KUKA KRL program: MyProgram_280().src

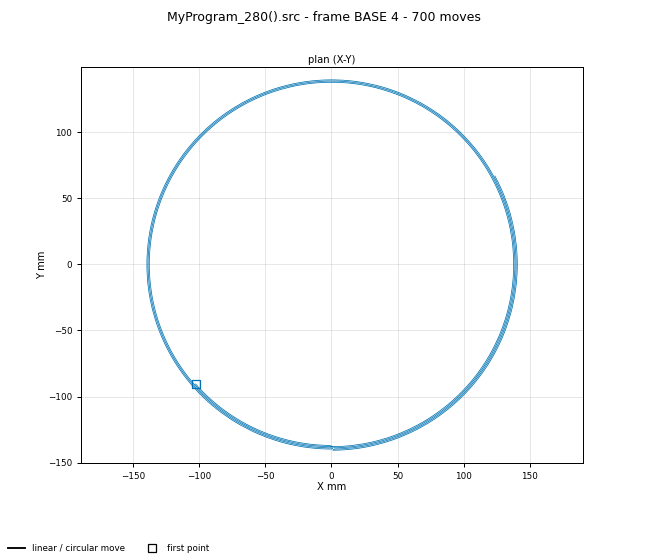
[picture p0: tool path of MyProgram_280().src in frame BASE 4, 700 of 700 moves have a stored position in this frame; points joined in program order, loops and branches not executed]
&ACCESS RVP
&REL 1
&PARAM TEMPLATE = C:\KRC\Roboter\Template\vorgabe
&PARAM EDITMASK = *
DEF MyProgram_280()
; ---- Setting reference (Base) ----
$BASE = BASE_DATA[4]

; --------------------------
; ---- Setting tool (TCP) ----
$TOOL = TOOL_DATA[3]
; --------------------------

$VEL.CP = VEL_APROX_PRINT
Startdeposition()
$VEL.CP = VEL_PRINT
LIN {X -102.883,Y -90.5499,Z 173,A -135.8281,B 8.3337,C 0.3369,E1 8.2218,E2 227.3937} C_DIS
LIN {X -99.9012,Y -93.8294,Z 173,A -133.9555,B 8.3335,C 0.3404,E1 8.2253,E2 225.5192} C_DIS
LIN {X -96.8965,Y -96.9297,Z 173,A -132.2443,B 8.3333,C 0.3455,E1 8.2287,E2 223.8206} C_DIS
LIN {X -93.9619,Y -99.7762,Z 173,A -130.464,B 8.3333,C 0.3476,E1 8.2323,E2 222.0316} C_DIS
LIN {X -90.696,Y -102.7539,Z 173,A -128.5932,B 8.3331,C 0.3506,E1 8.2362,E2 220.1583} C_DIS
LIN {X -87.7529,Y -105.2794,Z 173,A -126.8961,B 8.3331,C 0.3523,E1 8.2398,E2 218.452} C_DIS
LIN {X -84.2582,Y -108.0963,Z 173,A -125.0334,B 8.3329,C 0.3557,E1 8.2439,E2 216.5914} C_DIS
LIN {X -80.7877,Y -110.7143,Z 173,A -123.206,B 8.3328,C 0.3585,E1 8.248,E2 214.763} C_DIS
LIN {X -77.8003,Y -112.8331,Z 173,A -121.6319,B 8.3328,C 0.3602,E1 8.2516,E2 213.1836} C_DIS
LIN {X -74.2625,Y -115.1929,Z 173,A -119.9315,B 8.3325,C 0.3641,E1 8.2556,E2 211.4933} C_DIS
LIN {X -71.2942,Y -117.0532,Z 173,A -118.3313,B 8.3325,C 0.3639,E1 8.2594,E2 209.8758} C_DIS
LIN {X -67.4734,Y -119.2963,Z 173,A -116.5707,B 8.3324,C 0.368,E1 8.2636,E2 208.1271} C_DIS
LIN {X -64.4842,Y -120.9384,Z 173,A -115.1531,B 8.3323,C 0.3699,E1 8.2671,E2 206.7105} C_DIS
LIN {X -60.9886,Y -122.7359,Z 173,A -113.5525,B 8.3322,C 0.3726,E1 8.2711,E2 205.1153} C_DIS
LIN {X -57.8973,Y -124.2242,Z 173,A -112.0982,B 8.3322,C 0.3739,E1 8.2748,E2 203.6584} C_DIS
LIN {X -55.176,Y -125.4588,Z 173,A -110.7127,B 8.3322,C 0.3729,E1 8.2783,E2 202.2555} C_DIS
LIN {X -51.7787,Y -126.8971,Z 173,A -109.3505,B 8.332,C 0.3776,E1 8.2818,E2 200.9162} C_DIS
LIN {X -48.8661,Y -128.0485,Z 173,A -107.9192,B 8.332,C 0.3767,E1 8.2856,E2 199.4691} C_DIS
LIN {X -45.4055,Y -129.3145,Z 173,A -106.4697,B 8.3319,C 0.3796,E1 8.2893,E2 198.031} C_DIS
LIN {X -42.2502,Y -130.3796,Z 173,A -104.991,B 8.3319,C 0.3792,E1 8.2933,E2 196.541} C_DIS
LIN {X -39.0567,Y -131.3717,Z 173,A -103.5138,B 8.3319,C 0.3788,E1 8.2973,E2 195.0534} C_DIS
LIN {X -35.5511,Y -132.3624,Z 173,A -102.2773,B 8.3316,C 0.3849,E1 8.3005,E2 193.8532} C_DIS
LIN {X -32.916,Y -133.0445,Z 173,A -100.8373,B 8.3318,C 0.3802,E1 8.3045,E2 192.3743} C_DIS
LIN {X -29.7209,Y -133.7945,Z 173,A -99.4335,B 8.3318,C 0.3802,E1 8.3083,E2 190.966} C_DIS
LIN {X -25.9901,Y -134.5668,Z 173,A -98.0033,B 8.3317,C 0.3839,E1 8.3122,E2 189.5562} C_DIS
LIN {X -23.3494,Y -135.0523,Z 173,A -96.7469,B 8.3317,C 0.382,E1 8.3157,E2 188.2824} C_DIS
LIN {X -19.5757,Y -135.6484,Z 173,A -95.4567,B 8.3315,C 0.388,E1 8.3192,E2 187.0309} C_DIS
LIN {X -16.7714,Y -136.0246,Z 173,A -94.0487,B 8.3316,C 0.3842,E1 8.3231,E2 185.5937} C_DIS
LIN {X -13.2633,Y -136.4104,Z 173,A -92.8033,B 8.3314,C 0.3887,E1 8.3265,E2 184.3772} C_DIS
LIN {X -10.7558,Y -136.6332,Z 173,A -91.5229,B 8.3316,C 0.3847,E1 8.3302,E2 183.0672} C_DIS
LIN {X -7.653,Y -136.842,Z 173,A -90.2245,B 8.3316,C 0.3847,E1 8.3338,E2 181.7685} C_DIS
LIN {X -4.3301,Y -136.9863,Z 173,A -88.9268,B 8.3316,C 0.3865,E1 8.3374,E2 180.482} C_DIS
LIN {X -1.277,Y -137.0488,Z 173,A -87.465,B 8.3317,C 0.3829,E1 8.3415,E2 178.9959} C_DIS
LIN {X -1.277,Y -137.0488,Z 173,A -87.465,B 8.3317,C 0.3829,E1 8.3415,E2 178.9959} C_DIS
Enddeposition()
LIN {X 0.9792,Y -137.9557,Z 173,A -86.7312,B 8.287,C 0.3922,E1 8.2992,E2 178.3349} C_DIS
Startdeposition()
$VEL.CP = VEL_PRINT
LIN {X -2.0656,Y -137.947,Z 173,A -88.4524,B 8.2866,C 0.4008,E1 8.2942,E2 180.1156} C_DIS
LIN {X -5.8121,Y -137.8404,Z 173,A -89.9694,B 8.2866,C 0.4001,E1 8.29,E2 181.6282} C_DIS
LIN {X -9.6417,Y -137.6255,Z 173,A -91.5436,B 8.2866,C 0.3997,E1 8.2856,E2 183.2007} C_DIS
LIN {X -13.0454,Y -137.3441,Z 173,A -93.0201,B 8.2866,C 0.4006,E1 8.2815,E2 184.6851} C_DIS
LIN {X -16.3304,Y -136.9922,Z 173,A -94.7606,B 8.2863,C 0.407,E1 8.2765,E2 186.4732} C_DIS
LIN {X -20.1888,Y -136.4786,Z 173,A -95.9522,B 8.2867,C 0.3988,E1 8.2734,E2 187.6112} C_DIS
LIN {X -25.0424,Y -135.6715,Z 173,A -98.129,B 8.2867,C 0.4005,E1 8.2673,E2 189.8057} C_DIS
LIN {X -29.337,Y -134.8069,Z 173,A -99.8936,B 8.2867,C 0.3986,E1 8.2625,E2 191.5637} C_DIS
LIN {X -35.9245,Y -133.2031,Z 173,A -102.8001,B 8.2867,C 0.3986,E1 8.2546,E2 194.4825} C_DIS
LIN {X -39.9371,Y -132.0557,Z 173,A -104.3094,B 8.287,C 0.3934,E1 8.2506,E2 195.9636} C_DIS
LIN {X -43.1517,Y -131.0405,Z 173,A -105.8881,B 8.2869,C 0.3955,E1 8.2464,E2 197.5653} C_DIS
LIN {X -46.4079,Y -129.9228,Z 173,A -107.325,B 8.2869,C 0.3944,E1 8.2426,E2 199.0034} C_DIS
LIN {X -49.8097,Y -128.6564,Z 173,A -108.7224,B 8.2871,C 0.3911,E1 8.239,E2 200.3869} C_DIS
LIN {X -52.8849,Y -127.4234,Z 173,A -110.0787,B 8.2871,C 0.3894,E1 8.2355,E2 201.7409} C_DIS
LIN {X -55.7193,Y -126.2111,Z 173,A -111.6175,B 8.2871,C 0.3926,E1 8.2314,E2 203.3128} C_DIS
LIN {X -59.2158,Y -124.6074,Z 173,A -113.0992,B 8.2871,C 0.3888,E1 8.2277,E2 204.7798} C_DIS
LIN {X -62.027,Y -123.2334,Z 173,A -114.479,B 8.2871,C 0.3886,E1 8.2242,E2 206.1699} C_DIS
LIN {X -67.6249,Y -120.2533,Z 173,A -117.118,B 8.2873,C 0.3854,E1 8.2178,E2 208.8095} C_DIS
LIN {X -71.5832,Y -117.9401,Z 173,A -119.0316,B 8.2875,C 0.3829,E1 8.2132,E2 210.7242} C_DIS
LIN {X -75.3846,Y -115.5476,Z 173,A -120.9173,B 8.2875,C 0.3805,E1 8.2087,E2 212.6123} C_DIS
LIN {X -79.0785,Y -113.0517,Z 173,A -122.5617,B 8.2879,C 0.3742,E1 8.205,E2 214.2301} C_DIS
LIN {X -82.8628,Y -110.3079,Z 173,A -124.8045,B 8.2878,C 0.3761,E1 8.1999,E2 216.511} C_DIS
LIN {X -86.4464,Y -107.5223,Z 173,A -126.6718,B 8.2879,C 0.3725,E1 8.1958,E2 218.3757} C_DIS
LIN {X -89.7939,Y -104.7432,Z 173,A -128.5379,B 8.288,C 0.3703,E1 8.1918,E2 220.2489} C_DIS
LIN {X -93.0689,Y -101.8446,Z 173,A -130.3846,B 8.2882,C 0.3674,E1 8.1879,E2 222.099} C_DIS
LIN {X -96.4499,Y -98.648,Z 173,A -132.3135,B 8.2883,C 0.3636,E1 8.1841,E2 224.0269} C_DIS
LIN {X -99.3487,Y -95.7284,Z 173,A -133.9538,B 8.2885,C 0.3591,E1 8.1809,E2 225.658} C_DIS
LIN {X -102.0619,Y -92.8298,Z 173,A -135.8247,B 8.2885,C 0.3593,E1 8.1773,E2 227.5564} C_DIS
LIN {X -105.4509,Y -88.9619,Z 173,A -137.8991,B 8.2887,C 0.3538,E1 8.1735,E2 229.6222} C_DIS
LIN {X -108.3711,Y -85.3799,Z 173,A -139.8171,B 8.2889,C 0.3496,E1 8.1702,E2 231.5393} C_DIS
LIN {X -111.0969,Y -81.8015,Z 173,A -141.7145,B 8.2891,C 0.3458,E1 8.167,E2 233.4395} C_DIS
LIN {X -113.8226,Y -77.9641,Z 173,A -143.6412,B 8.2893,C 0.3408,E1 8.1639,E2 235.3618} C_DIS
LIN {X -116.0236,Y -74.6499,Z 173,A -145.3906,B 8.2893,C 0.3385,E1 8.1612,E2 237.1226} C_DIS
LIN {X -118.3482,Y -70.9068,Z 173,A -147.2546,B 8.2895,C 0.3346,E1 8.1585,E2 238.9899} C_DIS
LIN {X -120.7103,Y -66.8058,Z 173,A -148.9434,B 8.2899,C 0.3254,E1 8.1562,E2 240.6428} C_DIS
LIN {X -122.6542,Y -63.1648,Z 173,A -150.9243,B 8.2899,C 0.3252,E1 8.1536,E2 242.6563} C_DIS
LIN {X -124.3506,Y -59.7532,Z 173,A -152.4716,B 8.2901,C 0.3206,E1 8.1517,E2 244.1982} C_DIS
LIN {X -125.9172,Y -56.3763,Z 173,A -154.0438,B 8.2902,C 0.317,E1 8.1499,E2 245.7727} C_DIS
LIN {X -127.6592,Y -52.3184,Z 173,A -156.1711,B 8.2902,C 0.3167,E1 8.1476,E2 247.9356} C_DIS
LIN {X -129.6287,Y -47.2236,Z 173,A -158.1322,B 8.2906,C 0.306,E1 8.1457,E2 249.8567} C_DIS
LIN {X -131.0791,Y -43.0356,Z 173,A -160.2173,B 8.2906,C 0.3047,E1 8.1438,E2 251.9711} C_DIS
LIN {X -132.2357,Y -39.339,Z 173,A -161.6204,B 8.291,C 0.2972,E1 8.1426,E2 253.3474} C_DIS
LIN {X -133.2526,Y -35.7387,Z 173,A -163.1895,B 8.291,C 0.2931,E1 8.1415,E2 254.9171} C_DIS
LIN {X -134.083,Y -32.4849,Z 173,A -164.7412,B 8.2911,C 0.2916,E1 8.1404,E2 256.4875} C_DIS
LIN {X -134.8591,Y -29.0949,Z 173,A -166.1771,B 8.2913,C 0.2874,E1 8.1395,E2 257.9212} C_DIS
LIN {X -135.4963,Y -25.9666,Z 173,A -167.5733,B 8.2913,C 0.2847,E1 8.1388,E2 259.3251} C_DIS
LIN {X -136.1899,Y -22.0519,Z 173,A -169.348,B 8.2915,C 0.2819,E1 8.1379,E2 261.1141} C_DIS
LIN {X -136.7862,Y -17.9745,Z 173,A -170.9916,B 8.2917,C 0.276,E1 8.1373,E2 262.7477} C_DIS
LIN {X -137.1338,Y -15.0987,Z 173,A -172.2937,B 8.2917,C 0.274,E1 8.1369,E2 264.0611} C_DIS
LIN {X -137.5557,Y -10.5972,Z 173,A -174.1761,B 8.2919,C 0.2687,E1 8.1364,E2 265.9426} C_DIS
LIN {X -137.7677,Y -7.334,Z 173,A -175.3466,B 8.2921,C 0.262,E1 8.1362,E2 267.0885} C_DIS
LIN {X -137.9073,Y -3.8946,Z 173,A -176.7229,B 8.2923,C 0.2571,E1 8.1362,E2 268.4568} C_DIS
LIN {X -137.9604,Y -0.8702,Z 173,A -178.3723,B 8.2923,C 0.2593,E1 8.136,E2 270.1542} C_DIS
LIN {X -137.9142,Y 3.6454,Z 173,A 179.8464,B 8.2924,C 0.2525,E1 8.1361,E2 271.922} C_DIS
LIN {X -137.7534,Y 7.6193,Z 173,A 178.0993,B 8.2925,C 0.2491,E1 8.1364,E2 273.6796} C_DIS
LIN {X -137.5136,Y 11.1273,Z 173,A 176.677,B 8.2927,C 0.2444,E1 8.1367,E2 275.0958} C_DIS
LIN {X -137.266,Y 13.8585,Z 173,A 175.3981,B 8.2927,C 0.2432,E1 8.137,E2 276.391} C_DIS
LIN {X -136.7966,Y 17.8947,Z 173,A 173.84,B 8.2929,C 0.2364,E1 8.1375,E2 277.9314} C_DIS
LIN {X -136.2081,Y 21.9404,Z 173,A 171.938,B 8.2929,C 0.2345,E1 8.1384,E2 279.8571} C_DIS
LIN {X -135.5693,Y 25.5851,Z 173,A 170.1954,B 8.2929,C 0.2332,E1 8.1393,E2 281.6236} C_DIS
LIN {X -134.8756,Y 29.0186,Z 173,A 169.0835,B 8.2932,C 0.224,E1 8.1399,E2 282.6917} C_DIS
LIN {X -134.1832,Y 32.0691,Z 173,A 167.8519,B 8.2934,C 0.2193,E1 8.1406,E2 283.9137} C_DIS
LIN {X -133.5479,Y 34.626,Z 173,A 166.4523,B 8.2934,C 0.2208,E1 8.1416,E2 285.3501} C_DIS
LIN {X -132.4614,Y 38.568,Z 173,A 164.9416,B 8.2935,C 0.2133,E1 8.1428,E2 286.8359} C_DIS
LIN {X -131.4885,Y 41.7647,Z 173,A 163.4664,B 8.2935,C 0.2107,E1 8.144,E2 288.3205} C_DIS
LIN {X -130.3861,Y 45.0881,Z 173,A 162.0908,B 8.2937,C 0.2055,E1 8.1452,E2 289.685} C_DIS
LIN {X -129.4148,Y 47.8086,Z 173,A 160.87,B 8.2937,C 0.2026,E1 8.1464,E2 290.9072} C_DIS
LIN {X -128.0471,Y 51.356,Z 173,A 159.1779,B 8.2938,C 0.2,E1 8.1481,E2 292.6117} C_DIS
LIN {X -126.8766,Y 54.1862,Z 173,A 157.9737,B 8.2939,C 0.1956,E1 8.1494,E2 293.8063} C_DIS
LIN {X -125.338,Y 57.6533,Z 173,A 156.3034,B 8.294,C 0.1928,E1 8.1513,E2 295.4868} C_DIS
LIN {X -124.0777,Y 60.3222,Z 173,A 154.9133,B 8.294,C 0.1921,E1 8.153,E2 296.8959} C_DIS
LIN {X -122.3229,Y 63.8018,Z 173,A 153.4395,B 8.2942,C 0.1857,E1 8.1549,E2 298.3502} C_DIS
LIN {X -119.4454,Y 69.042,Z 173,A 150.8189,B 8.2942,C 0.1815,E1 8.1585,E2 300.9854} C_DIS
LIN {X -117.4741,Y 72.3455,Z 173,A 149.3691,B 8.2944,C 0.1753,E1 8.1605,E2 302.4155} C_DIS
LIN {X -115.4763,Y 75.4944,Z 173,A 147.5373,B 8.2944,C 0.1758,E1 8.1634,E2 304.2805} C_DIS
LIN {X -112.8589,Y 79.353,Z 173,A 145.5986,B 8.2944,C 0.1711,E1 8.1664,E2 306.2175} C_DIS
LIN {X -108.0056,Y 85.8415,Z 173,A 142.2322,B 8.2946,C 0.1634,E1 8.1721,E2 309.5808} C_DIS
LIN {X -105.3842,Y 89.0411,Z 173,A 140.4942,B 8.2947,C 0.1598,E1 8.1752,E2 311.3197} C_DIS
LIN {X -102.6871,Y 92.1376,Z 173,A 138.6772,B 8.2947,C 0.1578,E1 8.1786,E2 313.1487} C_DIS
LIN {X -99.6124,Y 95.4535,Z 173,A 136.8822,B 8.2948,C 0.1525,E1 8.182,E2 314.9317} C_DIS
LIN {X -96.9458,Y 98.1614,Z 173,A 135.2534,B 8.2948,C 0.1501,E1 8.1852,E2 316.5652} C_DIS
LIN {X -94.5977,Y 100.4254,Z 173,A 133.9095,B 8.2949,C 0.1472,E1 8.1879,E2 317.9065} C_DIS
LIN {X -91.4098,Y 103.3355,Z 173,A 132.0978,B 8.2949,C 0.144,E1 8.1917,E2 319.7189} C_DIS
LIN {X -88.4225,Y 105.9035,Z 173,A 130.3946,B 8.295,C 0.142,E1 8.1953,E2 321.4288} C_DIS
LIN {X -84.6977,Y 108.9051,Z 173,A 128.1797,B 8.295,C 0.142,E1 8.2003,E2 323.6698} C_DIS
LIN {X -82.0737,Y 110.8966,Z 173,A 126.9549,B 8.2951,C 0.1373,E1 8.203,E2 324.8759} C_DIS
LIN {X -78.2616,Y 113.6185,Z 173,A 125.0033,B 8.2951,C 0.1341,E1 8.2074,E2 326.8265} C_DIS
LIN {X -74.5584,Y 116.0821,Z 173,A 123.1927,B 8.2952,C 0.1306,E1 8.2116,E2 328.631} C_DIS
LIN {X -70.8901,Y 118.3582,Z 173,A 121.4157,B 8.2952,C 0.1276,E1 8.2159,E2 330.4046} C_DIS
LIN {X -66.2435,Y 121.0199,Z 173,A 119.0875,B 8.2952,C 0.1261,E1 8.2216,E2 332.7437} C_DIS
LIN {X -62.8343,Y 122.8224,Z 173,A 117.4404,B 8.2953,C 0.1247,E1 8.2256,E2 334.3949} C_DIS
LIN {X -58.5256,Y 124.9346,Z 173,A 115.4281,B 8.2953,C 0.1225,E1 8.2307,E2 336.4081} C_DIS
LIN {X -54.0934,Y 126.9167,Z 173,A 113.4525,B 8.2953,C 0.1195,E1 8.2358,E2 338.3772} C_DIS
LIN {X -50.0528,Y 128.5619,Z 173,A 111.7351,B 8.2954,C 0.1159,E1 8.2402,E2 340.0816} C_DIS
LIN {X -44.4017,Y 130.6241,Z 173,A 109.0787,B 8.2954,C 0.1161,E1 8.2472,E2 342.7556} C_DIS
LIN {X -40.5455,Y 131.8695,Z 173,A 107.5266,B 8.2954,C 0.1124,E1 8.2513,E2 344.2905} C_DIS
LIN {X -37.5348,Y 132.7583,Z 173,A 106.3779,B 8.2955,C 0.1087,E1 8.2543,E2 345.4192} C_DIS
LIN {X -34.2608,Y 133.6405,Z 173,A 104.8017,B 8.2955,C 0.1105,E1 8.2586,E2 347.0152} C_DIS
LIN {X -31.2296,Y 134.3819,Z 173,A 103.3807,B 8.2955,C 0.1118,E1 8.2625,E2 348.4506} C_DIS
LIN {X -27.6928,Y 135.1542,Z 173,A 102.1194,B 8.2955,C 0.1067,E1 8.2659,E2 349.6813} C_DIS
LIN {X -24.149,Y 135.8321,Z 173,A 100.5924,B 8.2955,C 0.1064,E1 8.2701,E2 351.2109} C_DIS
LIN {X -18.9902,Y 136.6499,Z 173,A 98.2921,B 8.2955,C 0.1077,E1 8.2765,E2 353.5262} C_DIS
LIN {X -15.1944,Y 137.1235,Z 173,A 96.2626,B 8.2955,C 0.1148,E1 8.2823,E2 355.6085} C_DIS
LIN {X -11.0614,Y 137.5191,Z 173,A 94.0381,B 8.2953,C 0.123,E1 8.2886,E2 357.8926} C_DIS
LIN {X -4.2782,Y 137.8966,Z 173,A 92.1554,B 8.2956,C 0.1063,E1 8.2936,E2 359.66} C_DIS
LIN {X 2.4377,Y 137.9408,Z 173,A 89.4986,B 8.2956,C 0.1039,E1 8.3009,E2 362.2993} C_DIS
LIN {X 9.6118,Y 137.6276,Z 173,A 86.5437,B 8.2956,C 0.1039,E1 8.3092,E2 365.2498} C_DIS
LIN {X 14.0894,Y 137.2425,Z 173,A 84.2938,B 8.2955,C 0.1112,E1 8.3156,E2 367.5462} C_DIS
LIN {X 17.8918,Y 136.797,Z 173,A 82.5683,B 8.2955,C 0.1142,E1 8.3204,E2 369.2876} C_DIS
LIN {X 21.6437,Y 136.2548,Z 173,A 81.2679,B 8.2955,C 0.1099,E1 8.3239,E2 370.5541} C_DIS
LIN {X 25.8341,Y 135.5216,Z 173,A 79.8227,B 8.2955,C 0.1049,E1 8.3277,E2 371.9592} C_DIS
LIN {X 28.7334,Y 134.9372,Z 173,A 77.9527,B 8.2955,C 0.1174,E1 8.3331,E2 373.9076} C_DIS
LIN {X 32.6672,Y 134.0391,Z 173,A 76.6406,B 8.2955,C 0.1118,E1 8.3365,E2 375.1749} C_DIS
LIN {X 36.9153,Y 132.9316,Z 173,A 75.1032,B 8.2955,C 0.1078,E1 8.3406,E2 376.6766} C_DIS
LIN {X 40.2181,Y 131.9697,Z 173,A 73.4973,B 8.2955,C 0.1123,E1 8.3449,E2 378.3042} C_DIS
LIN {X 43.4246,Y 130.9496,Z 173,A 72.0922,B 8.2955,C 0.1137,E1 8.3486,E2 379.71} C_DIS
LIN {X 46.7016,Y 129.8169,Z 173,A 70.6385,B 8.2955,C 0.1153,E1 8.3525,E2 381.1652} C_DIS
LIN {X 49.8442,Y 128.643,Z 173,A 69.3066,B 8.2955,C 0.1155,E1 8.3559,E2 382.4895} C_DIS
LIN {X 52.8129,Y 127.4535,Z 173,A 67.8602,B 8.2954,C 0.1192,E1 8.3597,E2 383.9503} C_DIS
LIN {X 56.2817,Y 125.9596,Z 173,A 66.4297,B 8.2954,C 0.1184,E1 8.3633,E2 385.3637} C_DIS
LIN {X 58.8172,Y 124.7978,Z 173,A 65.1493,B 8.2954,C 0.1221,E1 8.3666,E2 386.6592} C_DIS
LIN {X 64.1268,Y 122.1522,Z 173,A 62.8294,B 8.2954,C 0.1225,E1 8.3724,E2 388.9613} C_DIS
LIN {X 67.8596,Y 120.1214,Z 173,A 60.9316,B 8.2953,C 0.1276,E1 8.377,E2 390.8756} C_DIS
LIN {X 71.4457,Y 118.0233,Z 173,A 59.168,B 8.2953,C 0.1308,E1 8.3813,E2 392.644} C_DIS
LIN {X 75.4355,Y 115.5145,Z 173,A 56.7358,B 8.295,C 0.1431,E1 8.3871,E2 395.1347} C_DIS
LIN {X 79.858,Y 112.5026,Z 173,A 55.1002,B 8.2951,C 0.1353,E1 8.3907,E2 396.6986} C_DIS
LIN {X 83.4863,Y 109.837,Z 173,A 53.2184,B 8.2951,C 0.1387,E1 8.3949,E2 398.5822} C_DIS
LIN {X 87.0974,Y 106.9957,Z 173,A 51.3463,B 8.2951,C 0.1414,E1 8.399,E2 400.4502} C_DIS
LIN {X 90.4066,Y 104.2151,Z 173,A 49.7304,B 8.2951,C 0.1412,E1 8.4023,E2 402.0444} C_DIS
LIN {X 92.9479,Y 101.9548,Z 173,A 48.199,B 8.295,C 0.1463,E1 8.4056,E2 403.5909} C_DIS
LIN {X 95.0442,Y 100.0037,Z 173,A 46.8658,B 8.2949,C 0.1515,E1 8.4083,E2 404.9422} C_DIS
LIN {X 98.5503,Y 96.5496,Z 173,A 44.3971,B 8.2946,C 0.1642,E1 8.4133,E2 407.4639} C_DIS
LIN {X 102.3654,Y 92.4953,Z 173,A 42.7347,B 8.2948,C 0.156,E1 8.4162,E2 409.0471} C_DIS
LIN {X 105.1615,Y 89.303,Z 173,A 41.0308,B 8.2948,C 0.1586,E1 8.4193,E2 410.7443} C_DIS
LIN {X 107.7501,Y 86.1625,Z 173,A 39.4496,B 8.2948,C 0.1602,E1 8.4221,E2 412.3126} C_DIS
LIN {X 110.3043,Y 82.8676,Z 173,A 37.602,B 8.2946,C 0.1665,E1 8.4252,E2 414.1755} C_DIS
LIN {X 112.8049,Y 79.4295,Z 173,A 35.8745,B 8.2946,C 0.1698,E1 8.428,E2 415.8991} C_DIS
LIN {X 115.6759,Y 75.1869,Z 173,A 33.7901,B 8.2944,C 0.174,E1 8.4313,E2 417.9791} C_DIS
LIN {X 117.6682,Y 72.0291,Z 173,A 31.4583,B 8.294,C 0.1939,E1 8.4348,E2 420.4085} C_DIS
LIN {X 120.956,Y 66.3608,Z 173,A 29.5461,B 8.2942,C 0.184,E1 8.4373,E2 422.2221} C_DIS
LIN {X 122.8108,Y 62.8571,Z 173,A 28.056,B 8.2942,C 0.1849,E1 8.4392,E2 423.6936} C_DIS
LIN {X 124.0311,Y 60.4167,Z 173,A 26.7856,B 8.2941,C 0.1907,E1 8.4408,E2 424.9818} C_DIS
LIN {X 125.8177,Y 56.5988,Z 173,A 25.148,B 8.2941,C 0.1929,E1 8.4426,E2 426.6064} C_DIS
LIN {X 127.1655,Y 53.5024,Z 173,A 23.5644,B 8.2938,C 0.2004,E1 8.4444,E2 428.2135} C_DIS
LIN {X 129.0833,Y 48.6934,Z 173,A 21.8115,B 8.2938,C 0.1979,E1 8.4461,E2 429.9182} C_DIS
LIN {X 130.2557,Y 45.4643,Z 173,A 20.3126,B 8.2938,C 0.2033,E1 8.4476,E2 431.4271} C_DIS
LIN {X 131.3571,Y 42.176,Z 173,A 18.8517,B 8.2937,C 0.2076,E1 8.4488,E2 432.8916} C_DIS
LIN {X 132.4689,Y 38.5423,Z 173,A 17.3109,B 8.2936,C 0.2112,E1 8.4501,E2 434.4289} C_DIS
LIN {X 133.5496,Y 34.6192,Z 173,A 15.7227,B 8.2936,C 0.2137,E1 8.4512,E2 436.0056} C_DIS
LIN {X 134.2706,Y 31.7066,Z 173,A 14.363,B 8.2934,C 0.2196,E1 8.4521,E2 437.3805} C_DIS
LIN {X 135.3757,Y 26.5975,Z 173,A 12.2298,B 8.2932,C 0.225,E1 8.4533,E2 439.5108} C_DIS
LIN {X 136.0321,Y 22.9972,Z 173,A 10.7781,B 8.2932,C 0.2278,E1 8.454,E2 440.9551} C_DIS
LIN {X 136.4964,Y 20.0641,Z 173,A 9.58,B 8.2931,C 0.2306,E1 8.4545,E2 442.1497} C_DIS
LIN {X 136.9545,Y 16.6463,Z 173,A 8.332,B 8.2931,C 0.2308,E1 8.455,E2 443.3757} C_DIS
LIN {X 137.4651,Y 11.7013,Z 173,A 6.3071,B 8.2929,C 0.2359,E1 8.4555,E2 445.3974} C_DIS
LIN {X 137.8923,Y 4.4322,Z 173,A 2.4349,B 8.2921,C 0.2626,E1 8.456,E2 449.3788} C_DIS
LIN {X 137.9561,Y -1.5094,Z 173,A 0.8012,B 8.2924,C 0.2521,E1 8.456,E2 450.9101} C_DIS
LIN {X 137.657,Y -9.1992,Z 173,A -2.2907,B 8.2922,C 0.2591,E1 8.4557,E2 453.9919} C_DIS
LIN {X 136.9661,Y -16.5491,Z 173,A -4.9984,B 8.2922,C 0.2603,E1 8.455,E2 456.657} C_DIS
LIN {X 136.1629,Y -22.2132,Z 173,A -7.9334,B 8.2916,C 0.2791,E1 8.4537,E2 459.6656} C_DIS
LIN {X 135.038,Y -28.2635,Z 173,A -10.2159,B 8.2916,C 0.2806,E1 8.4525,E2 461.9159} C_DIS
LIN {X 134.3943,Y -31.1752,Z 173,A -11.5694,B 8.2913,C 0.2866,E1 8.4517,E2 463.2852} C_DIS
LIN {X 133.5485,Y -34.6235,Z 173,A -12.9835,B 8.2913,C 0.2895,E1 8.4507,E2 464.6932} C_DIS
LIN {X 132.6447,Y -37.9395,Z 173,A -14.4161,B 8.2911,C 0.2936,E1 8.4496,E2 466.1278} C_DIS
LIN {X 131.5129,Y -41.6883,Z 173,A -15.9147,B 8.2911,C 0.2954,E1 8.4484,E2 467.6118} C_DIS
LIN {X 130.3865,Y -45.087,Z 173,A -17.3284,B 8.2909,C 0.2979,E1 8.4471,E2 469.0177} C_DIS
LIN {X 129.4055,Y -47.8333,Z 173,A -18.4578,B 8.2909,C 0.2995,E1 8.4461,E2 470.1379} C_DIS
LIN {X 127.8905,Y -51.7446,Z 173,A -20.2536,B 8.2907,C 0.3054,E1 8.4442,E2 471.9424} C_DIS
LIN {X 126.6647,Y -54.6763,Z 173,A -21.5571,B 8.2905,C 0.3086,E1 8.4428,E2 473.2451} C_DIS
LIN {X 123.554,Y -61.3839,Z 173,A -24.5387,B 8.2903,C 0.3149,E1 8.4393,E2 476.2185} C_DIS
LIN {X 121.8158,Y -64.7676,Z 173,A -26.1934,B 8.2901,C 0.3206,E1 8.4371,E2 477.8844} C_DIS
LIN {X 119.8061,Y -68.414,Z 173,A -27.9228,B 8.2899,C 0.3251,E1 8.4348,E2 479.6156} C_DIS
LIN {X 117.8429,Y -71.7423,Z 173,A -29.9468,B 8.2894,C 0.3379,E1 8.4318,E2 481.6946} C_DIS
LIN {X 115.366,Y -75.6618,Z 173,A -31.3709,B 8.2896,C 0.3322,E1 8.4297,E2 483.0569} C_DIS
LIN {X 113.106,Y -79.0005,Z 173,A -32.9855,B 8.2896,C 0.335,E1 8.4271,E2 484.6655} C_DIS
LIN {X 110.7876,Y -82.22,Z 173,A -34.5935,B 8.2894,C 0.3382,E1 8.4245,E2 486.2702} C_DIS
LIN {X 107.439,Y -86.5497,Z 173,A -36.9137,B 8.2891,C 0.3445,E1 8.4205,E2 488.5987} C_DIS
LIN {X 104.8112,Y -89.7149,Z 173,A -38.6292,B 8.289,C 0.3485,E1 8.4174,E2 490.3168} C_DIS
LIN {X 102.4431,Y -92.4097,Z 173,A -40.926,B 8.2881,C 0.3685,E1 8.4129,E2 492.7174} C_DIS
LIN {X 97.7231,Y -97.387,Z 173,A -42.6543,B 8.2888,C 0.3515,E1 8.4098,E2 494.3062} C_DIS
LIN {X 92.825,Y -102.0663,Z 173,A -45.9549,B 8.2882,C 0.3673,E1 8.403,E2 497.6718} C_DIS
LIN {X 90.0018,Y -104.5639,Z 173,A -47.4217,B 8.2882,C 0.3684,E1 8.3999,E2 499.1276} C_DIS
LIN {X 87.4209,Y -106.7314,Z 173,A -48.5305,B 8.2882,C 0.3652,E1 8.3976,E2 500.2006} C_DIS
LIN {X 80.5503,Y -112.0076,Z 173,A -52.2363,B 8.2879,C 0.374,E1 8.3893,E2 503.9236} C_DIS
LIN {X 76.5129,Y -114.8032,Z 173,A -54.1437,B 8.2879,C 0.3748,E1 8.3849,E2 505.8159} C_DIS
LIN {X 72.2616,Y -117.5256,Z 173,A -56.4554,B 8.2875,C 0.3825,E1 8.3794,E2 508.1569} C_DIS
LIN {X 69.3793,Y -119.2501,Z 173,A -57.651,B 8.2875,C 0.3807,E1 8.3765,E2 509.3283} C_DIS
LIN {X 65.4205,Y -121.4667,Z 173,A -59.5615,B 8.2875,C 0.3841,E1 8.3718,E2 511.2438} C_DIS
LIN {X 61.4938,Y -123.4998,Z 173,A -61.2232,B 8.2875,C 0.3832,E1 8.3678,E2 512.8846} C_DIS
LIN {X 58.8169,Y -124.798,Z 173,A -62.6357,B 8.2872,C 0.3884,E1 8.3641,E2 514.3209} C_DIS
LIN {X 52.5865,Y -127.548,Z 173,A -65.1704,B 8.2873,C 0.3861,E1 8.3577,E2 516.8201} C_DIS
LIN {X 47.5517,Y -129.5104,Z 173,A -67.5563,B 8.2871,C 0.3915,E1 8.3515,E2 519.226} C_DIS
LIN {X 42.1045,Y -131.38,Z 173,A -69.8552,B 8.2871,C 0.3921,E1 8.3454,E2 521.5147} C_DIS
LIN {X 39.0329,Y -132.3253,Z 173,A -71.1777,B 8.287,C 0.3932,E1 8.3419,E2 522.8366} C_DIS
LIN {X 36.1751,Y -133.1363,Z 173,A -72.5335,B 8.2868,C 0.3966,E1 8.3382,E2 524.209} C_DIS
LIN {X 31.3763,Y -134.3483,Z 173,A -74.5549,B 8.2868,C 0.3976,E1 8.3327,E2 526.2273} C_DIS
LIN {X 27.4863,Y -135.1962,Z 173,A -75.9085,B 8.287,C 0.393,E1 8.3291,E2 527.5435} C_DIS
LIN {X 24.6497,Y -135.7425,Z 173,A -77.4053,B 8.2867,C 0.3995,E1 8.3249,E2 529.0792} C_DIS
LIN {X 16.0145,Y -137.0299,Z 173,A -81.034,B 8.2866,C 0.4015,E1 8.3149,E2 532.7105} C_DIS
LIN {X 11.9861,Y -137.441,Z 173,A -82.6646,B 8.2866,C 0.4012,E1 8.3103,E2 534.3354} C_DIS
LIN {X 7.7255,Y -137.7478,Z 173,A -84.4968,B 8.2866,C 0.4028,E1 8.3052,E2 536.1761} C_DIS
LIN {X 4.1448,Y -137.9003,Z 173,A -85.8866,B 8.2866,C 0.4013,E1 8.3013,E2 537.554} C_DIS
LIN {X 0.9792,Y -137.9557,Z 173,A -86.7279,B 8.287,C 0.3927,E1 8.2992,E2 538.3348} C_DIS
Enddeposition()
LIN {X 0.9792,Y -137.9557,Z 173,A -86.7279,B 8.287,C 0.3927,E1 8.2992,E2 538.3348} C_DIS
Startdeposition()
$VEL.CP = VEL_PRINT
LIN {X 2.7915,Y -138.8436,Z 173,A -85.7711,B 8.2411,C 0.3941,E1 8.256,E2 537.3975} C_DIS
LIN {X 6.4638,Y -138.7212,Z 173,A -84.1933,B 8.2411,C 0.3925,E1 8.2604,E2 535.8108} C_DIS
LIN {X 10.1394,Y -138.5001,Z 173,A -82.7319,B 8.2411,C 0.3932,E1 8.2645,E2 534.3561} C_DIS
LIN {X 13.6741,Y -138.1964,Z 173,A -81.1883,B 8.2412,C 0.3911,E1 8.2688,E2 532.8013} C_DIS
LIN {X 18.8142,Y -137.5924,Z 173,A -78.6523,B 8.2416,C 0.3823,E1 8.276,E2 530.2114} C_DIS
LIN {X 22.9677,Y -136.9581,Z 173,A -77.0567,B 8.2416,C 0.3839,E1 8.2803,E2 528.6328} C_DIS
LIN {X 26.6001,Y -136.3002,Z 173,A -75.9155,B 8.2413,C 0.3904,E1 8.2833,E2 527.5409} C_DIS
LIN {X 30.0295,Y -135.5868,Z 173,A -73.8541,B 8.2419,C 0.3772,E1 8.2892,E2 525.3975} C_DIS
LIN {X 34.8677,Y -134.4238,Z 173,A -72.4296,B 8.2414,C 0.3879,E1 8.2928,E2 524.0543} C_DIS
LIN {X 38.0658,Y -133.5532,Z 173,A -70.9272,B 8.2416,C 0.384,E1 8.2969,E2 522.5333} C_DIS
LIN {X 41.9588,Y -132.3803,Z 173,A -69.0938,B 8.2418,C 0.3793,E1 8.3018,E2 520.6782} C_DIS
LIN {X 45.0896,Y -131.3472,Z 173,A -67.8535,B 8.2418,C 0.3803,E1 8.3051,E2 519.4527} C_DIS
LIN {X 49.7627,Y -129.6495,Z 173,A -66.0832,B 8.2416,C 0.3836,E1 8.3096,E2 517.7177} C_DIS
LIN {X 52.678,Y -128.4938,Z 173,A -64.4049,B 8.242,C 0.3743,E1 8.3141,E2 515.988} C_DIS
LIN {X 55.6978,Y -127.2129,Z 173,A -63.2244,B 8.242,C 0.3761,E1 8.317,E2 514.8291} C_DIS
LIN {X 60.1844,Y -125.1515,Z 173,A -61.2903,B 8.242,C 0.3755,E1 8.3219,E2 512.9067} C_DIS
LIN {X 63.4522,Y -123.5274,Z 173,A -59.7786,B 8.242,C 0.3732,E1 8.3257,E2 511.3931} C_DIS
LIN {X 67.5973,Y -121.3105,Z 173,A -57.8518,B 8.2422,C 0.3706,E1 8.3304,E2 509.4664} C_DIS
LIN {X 74.5256,Y -117.1819,Z 173,A -54.5543,B 8.2424,C 0.3659,E1 8.3383,E2 506.1701} C_DIS
LIN {X 78.0932,Y -114.8348,Z 173,A -52.2595,B 8.243,C 0.3519,E1 8.3437,E2 503.8035} C_DIS
LIN {X 82.3148,Y -111.8471,Z 173,A -50.7958,B 8.2426,C 0.362,E1 8.3469,E2 502.426} C_DIS
LIN {X 85.988,Y -109.0487,Z 173,A -49.0413,B 8.2426,C 0.3616,E1 8.3507,E2 500.6895} C_DIS
LIN {X 88.3689,Y -107.1284,Z 173,A -46.9626,B 8.2434,C 0.3421,E1 8.3554,E2 498.5023} C_DIS
LIN {X 92.5328,Y -103.5529,Z 173,A -45.3364,B 8.243,C 0.351,E1 8.3586,E2 496.958} C_DIS
LIN {X 95.8393,Y -100.5005,Z 173,A -43.5723,B 8.2431,C 0.3491,E1 8.3622,E2 495.2043} C_DIS
LIN {X 98.7491,Y -97.6433,Z 173,A -41.2737,B 8.2438,C 0.3325,E1 8.3669,E2 492.8231} C_DIS
LIN {X 102.3649,Y -93.8452,Z 173,A -39.7632,B 8.2434,C 0.3416,E1 8.3696,E2 491.3963} C_DIS
LIN {X 106.6199,Y -88.9821,Z 173,A -37.1608,B 8.2436,C 0.3369,E1 8.3744,E2 488.7997} C_DIS
LIN {X 109.7793,Y -85.0527,Z 173,A -34.9231,B 8.2439,C 0.3288,E1 8.3783,E2 486.5392} C_DIS
LIN {X 112.6169,Y -81.2589,Z 173,A -33.3124,B 8.2439,C 0.3314,E1 8.3809,E2 484.9715} C_DIS
LIN {X 114.5324,Y -78.5355,Z 173,A -31.7365,B 8.2441,C 0.3238,E1 8.3834,E2 483.3678} C_DIS
LIN {X 117.6555,Y -73.7754,Z 173,A -29.3658,B 8.2444,C 0.3175,E1 8.387,E2 480.992} C_DIS
LIN {X 119.6122,Y -70.5583,Z 173,A -27.8851,B 8.2444,C 0.3151,E1 8.3891,E2 479.5192} C_DIS
LIN {X 121.7969,Y -66.7164,Z 173,A -26.0602,B 8.2446,C 0.3104,E1 8.3916,E2 477.6923} C_DIS
LIN {X 124.274,Y -61.9781,Z 173,A -24.0977,B 8.2446,C 0.3098,E1 8.3941,E2 475.7591} C_DIS
LIN {X 128.1029,Y -53.6155,Z 173,A -20.5421,B 8.2448,C 0.3049,E1 8.3982,E2 472.231} C_DIS
LIN {X 130.1071,Y -48.5503,Z 173,A -18.0246,B 8.2453,C 0.2929,E1 8.4007,E2 469.6764} C_DIS
LIN {X 131.3033,Y -45.216,Z 173,A -16.6116,B 8.2453,C 0.2899,E1 8.402,E2 468.2682} C_DIS
LIN {X 132.3085,Y -42.1835,Z 173,A -15.2854,B 8.2455,C 0.2861,E1 8.4032,E2 466.9397} C_DIS
LIN {X 133.9637,Y -36.5975,Z 173,A -12.7731,B 8.2458,C 0.277,E1 8.4051,E2 464.411} C_DIS
LIN {X 134.9341,Y -32.8311,Z 173,A -11.3133,B 8.2458,C 0.2756,E1 8.4061,E2 462.9684} C_DIS
LIN {X 135.8619,Y -28.7555,Z 173,A -9.0496,B 8.2464,C 0.259,E1 8.4075,E2 460.6328} C_DIS
LIN {X 136.8671,Y -23.5132,Z 173,A -7.5976,B 8.2461,C 0.269,E1 8.4081,E2 459.2763} C_DIS
LIN {X 137.4451,Y -19.8477,Z 173,A -6.2593,B 8.2461,C 0.2688,E1 8.4087,E2 457.9614} C_DIS
LIN {X 138.0126,Y -15.4246,Z 173,A -3.5904,B 8.2468,C 0.2455,E1 8.4096,E2 455.1832} C_DIS
LIN {X 138.4893,Y -10.2868,Z 173,A -2.1849,B 8.2465,C 0.2551,E1 8.4099,E2 453.8697} C_DIS
LIN {X 138.8103,Y -4.1053,Z 173,A 0.1651,B 8.2466,C 0.2521,E1 8.4102,E2 451.5437} C_DIS
LIN {X 138.8731,Y -0.2305,Z 173,A 2.4441,B 8.2472,C 0.2328,E1 8.4102,E2 449.1754} C_DIS
LIN {X 138.8115,Y 4.0627,Z 173,A 4.2319,B 8.2473,C 0.2273,E1 8.4101,E2 447.3839} C_DIS
LIN {X 138.594,Y 8.766,Z 173,A 5.6092,B 8.2472,C 0.2339,E1 8.4099,E2 446.0781} C_DIS
LIN {X 138.278,Y 12.8241,Z 173,A 7.9361,B 8.2477,C 0.2151,E1 8.4093,E2 443.6659} C_DIS
LIN {X 137.6625,Y 18.2796,Z 173,A 9.2767,B 8.2473,C 0.2286,E1 8.4088,E2 442.4429} C_DIS
LIN {X 137.226,Y 21.3089,Z 173,A 10.7357,B 8.2475,C 0.2208,E1 8.4082,E2 440.9578} C_DIS
LIN {X 136.6711,Y 24.6181,Z 173,A 12.0908,B 8.2475,C 0.2175,E1 8.4076,E2 439.6053} C_DIS
LIN {X 135.3282,Y 31.1666,Z 173,A 14.7958,B 8.2478,C 0.2108,E1 8.406,E2 436.905} C_DIS
LIN {X 134.4087,Y 34.9275,Z 173,A 16.4494,B 8.2479,C 0.2052,E1 8.4049,E2 435.2431} C_DIS
LIN {X 133.3461,Y 38.7796,Z 173,A 18.035,B 8.2479,C 0.202,E1 8.4037,E2 433.6642} C_DIS
LIN {X 132.3215,Y 42.1427,Z 173,A 19.4078,B 8.248,C 0.1996,E1 8.4025,E2 432.3004} C_DIS
LIN {X 131.1875,Y 45.5501,Z 173,A 20.869,B 8.2481,C 0.196,E1 8.4012,E2 430.8407} C_DIS
LIN {X 129.9184,Y 49.0542,Z 173,A 22.423,B 8.2482,C 0.1915,E1 8.3997,E2 429.2837} C_DIS
LIN {X 127.3285,Y 55.4303,Z 173,A 25.0758,B 8.2483,C 0.188,E1 8.3969,E2 426.6529} C_DIS
LIN {X 126.1535,Y 58.0544,Z 173,A 26.6038,B 8.2485,C 0.1776,E1 8.3951,E2 425.0805} C_DIS
LIN {X 124.7686,Y 60.9753,Z 173,A 27.531,B 8.2485,C 0.1828,E1 8.394,E2 424.2044} C_DIS
LIN {X 123.562,Y 63.3842,Z 173,A 28.7701,B 8.2485,C 0.1772,E1 8.3924,E2 422.9484} C_DIS
LIN {X 121.7346,Y 66.8306,Z 173,A 30.8832,B 8.2489,C 0.1626,E1 8.3895,E2 420.77} C_DIS
LIN {X 119.4032,Y 70.9096,Z 173,A 32.6245,B 8.2489,C 0.1619,E1 8.3871,E2 419.0529} C_DIS
LIN {X 117.3715,Y 74.2256,Z 173,A 33.5303,B 8.2487,C 0.1727,E1 8.3859,E2 418.2354} C_DIS
LIN {X 114.6436,Y 78.3735,Z 173,A 35.9045,B 8.2489,C 0.161,E1 8.3821,E2 415.8188} C_DIS
LIN {X 112.1678,Y 81.8783,Z 173,A 37.7211,B 8.2489,C 0.1559,E1 8.3792,E2 413.9955} C_DIS
LIN {X 108.1155,Y 87.1581,Z 173,A 40.1744,B 8.2489,C 0.1558,E1 8.375,E2 411.5783} C_DIS
LIN {X 106.1467,Y 89.5461,Z 173,A 41.6346,B 8.2491,C 0.1492,E1 8.3724,E2 410.0944} C_DIS
LIN {X 103.431,Y 92.6689,Z 173,A 44.0753,B 8.2494,C 0.1304,E1 8.3676,E2 407.5593} C_DIS
LIN {X 99.0933,Y 97.2934,Z 173,A 45.7114,B 8.2492,C 0.1452,E1 8.3647,E2 406.0474} C_DIS
LIN {X 96.5951,Y 99.7735,Z 173,A 47.4901,B 8.2493,C 0.1356,E1 8.3611,E2 404.227} C_DIS
LIN {X 93.257,Y 102.9011,Z 173,A 49.1809,B 8.2493,C 0.1359,E1 8.3576,E2 402.5606} C_DIS
LIN {X 90.93,Y 104.9637,Z 173,A 50.4384,B 8.2493,C 0.134,E1 8.355,E2 401.3061} C_DIS
LIN {X 87.606,Y 107.7535,Z 173,A 52.2706,B 8.2494,C 0.1299,E1 8.351,E2 399.4682} C_DIS
LIN {X 84.0746,Y 110.5309,Z 173,A 54.0936,B 8.2494,C 0.1273,E1 8.347,E2 397.6487} C_DIS
LIN {X 80.4866,Y 113.1704,Z 173,A 56.1378,B 8.2496,C 0.1201,E1 8.3423,E2 395.578} C_DIS
LIN {X 77.6549,Y 115.131,Z 173,A 57.4254,B 8.2496,C 0.1205,E1 8.3394,E2 394.3072} C_DIS
LIN {X 74.5876,Y 117.1422,Z 173,A 58.817,B 8.2496,C 0.1205,E1 8.3361,E2 392.9308} C_DIS
LIN {X 71.5973,Y 118.9934,Z 173,A 60.0683,B 8.2496,C 0.1224,E1 8.3332,E2 391.7047} C_DIS
LIN {X 68.5797,Y 120.7576,Z 173,A 61.6829,B 8.2496,C 0.1169,E1 8.3293,E2 390.0683} C_DIS
LIN {X 64.8314,Y 122.8084,Z 173,A 64.3545,B 8.2499,C 0.0966,E1 8.3224,E2 387.2809} C_DIS
LIN {X 58.2768,Y 126.0506,Z 173,A 66.3074,B 8.2497,C 0.1138,E1 8.3178,E2 385.4634} C_DIS
LIN {X 55.2723,Y 127.3968,Z 173,A 68.0345,B 8.2497,C 0.1051,E1 8.3132,E2 383.69} C_DIS
LIN {X 51.8972,Y 128.8085,Z 173,A 69.2102,B 8.2497,C 0.1099,E1 8.3103,E2 382.5565} C_DIS
LIN {X 48.7081,Y 130.048,Z 173,A 70.5999,B 8.2497,C 0.1089,E1 8.3067,E2 381.1696} C_DIS
LIN {X 45.3433,Y 131.2592,Z 173,A 72.0556,B 8.2497,C 0.1079,E1 8.3029,E2 379.7166} C_DIS
LIN {X 41.9909,Y 132.37,Z 173,A 73.501,B 8.2497,C 0.1069,E1 8.299,E2 378.273} C_DIS
LIN {X 38.6917,Y 133.3719,Z 173,A 74.9231,B 8.2497,C 0.1057,E1 8.2952,E2 376.8512} C_DIS
LIN {X 35.5213,Y 134.2509,Z 173,A 76.296,B 8.2497,C 0.1044,E1 8.2915,E2 375.4766} C_DIS
LIN {X 26.0914,Y 136.3974,Z 173,A 79.9338,B 8.2497,C 0.1086,E1 8.2818,E2 371.8842} C_DIS
LIN {X 20.3432,Y 137.3733,Z 173,A 82.8602,B 8.2499,C 0.0979,E1 8.2735,E2 368.8935} C_DIS
LIN {X 12.5514,Y 138.3042,Z 173,A 85.8416,B 8.2499,C 0.1016,E1 8.2653,E2 365.9454} C_DIS
LIN {X 9.1313,Y 138.5715,Z 173,A 87.8166,B 8.2499,C 0.0911,E1 8.2596,E2 363.9006} C_DIS
LIN {X 4.5135,Y 138.7988,Z 173,A 89.3654,B 8.2499,C 0.0975,E1 8.2554,E2 362.3979} C_DIS
LIN {X 0.1081,Y 138.8724,Z 173,A 90.9512,B 8.2499,C 0.1016,E1 8.2511,E2 360.8419} C_DIS
LIN {X -2.6947,Y 138.8452,Z 173,A 92.2163,B 8.2499,C 0.0997,E1 8.2475,E2 359.5637} C_DIS
LIN {X -9.8843,Y 138.5187,Z 173,A 94.939,B 8.2498,C 0.1046,E1 8.24,E2 356.8734} C_DIS
LIN {X -17.1416,Y 137.8104,Z 173,A 98.1352,B 8.2498,C 0.1023,E1 8.2311,E2 353.6557} C_DIS
LIN {X -22.0587,Y 137.1091,Z 173,A 100.3812,B 8.2498,C 0.0997,E1 8.2248,E2 351.3863} C_DIS
LIN {X -26.669,Y 136.287,Z 173,A 102.1342,B 8.2498,C 0.1039,E1 8.22,E2 349.6569} C_DIS
LIN {X -30.0886,Y 135.5741,Z 173,A 103.5841,B 8.2498,C 0.1046,E1 8.2161,E2 348.2068} C_DIS
LIN {X -33.0206,Y 134.8884,Z 173,A 104.9725,B 8.2498,C 0.103,E1 8.2123,E2 346.8009} C_DIS
LIN {X -37.3154,Y 133.7631,Z 173,A 106.7064,B 8.2498,C 0.106,E1 8.2076,E2 345.0804} C_DIS
LIN {X -40.8036,Y 132.7406,Z 173,A 108.1928,B 8.2498,C 0.1075,E1 8.2036,E2 343.5968} C_DIS
LIN {X -44.5347,Y 131.5375,Z 173,A 110.0709,B 8.2498,C 0.1046,E1 8.1986,E2 341.6872} C_DIS
LIN {X -50.1114,Y 129.5139,Z 173,A 112.3765,B 8.2498,C 0.1095,E1 8.1926,E2 339.4012} C_DIS
LIN {X -54.2488,Y 127.8384,Z 173,A 114.1369,B 8.2497,C 0.1129,E1 8.1881,E2 337.6524} C_DIS
LIN {X -57.93,Y 126.211,Z 173,A 116.3119,B 8.2497,C 0.1063,E1 8.1824,E2 335.4141} C_DIS
LIN {X -61.9769,Y 124.2746,Z 173,A 117.6737,B 8.2497,C 0.1169,E1 8.1792,E2 334.1152} C_DIS
LIN {X -65.1076,Y 122.6634,Z 173,A 119.1682,B 8.2497,C 0.1182,E1 8.1754,E2 332.6167} C_DIS
LIN {X -72.3442,Y 118.5408,Z 173,A 122.4084,B 8.2495,C 0.1264,E1 8.1677,E2 329.4041} C_DIS
LIN {X -75.5899,Y 116.4975,Z 173,A 124.0664,B 8.2495,C 0.1277,E1 8.1637,E2 327.738} C_DIS
LIN {X -78.2403,Y 114.735,Z 173,A 125.6449,B 8.2495,C 0.1255,E1 8.16,E2 326.1275} C_DIS
LIN {X -81.8701,Y 112.1738,Z 173,A 128.1644,B 8.2496,C 0.1175,E1 8.1541,E2 323.5231} C_DIS
LIN {X -86.5544,Y 108.5994,Z 173,A 129.758,B 8.2493,C 0.1354,E1 8.1509,E2 322.0372} C_DIS
LIN {X -89.4651,Y 106.2147,Z 173,A 131.5271,B 8.2493,C 0.1348,E1 8.147,E2 320.2425} C_DIS
LIN {X -94.0099,Y 102.2136,Z 173,A 134.3306,B 8.2493,C 0.1348,E1 8.1411,E2 317.4029} C_DIS
LIN {X -96.7883,Y 99.5871,Z 173,A 135.4443,B 8.2492,C 0.1454,E1 8.139,E2 316.349} C_DIS
LIN {X -99.302,Y 97.0807,Z 173,A 137.1256,B 8.2492,C 0.145,E1 8.1356,E2 314.6419} C_DIS
LIN {X -103.5765,Y 92.5064,Z 173,A 139.8539,B 8.2492,C 0.1483,E1 8.1305,E2 311.8979} C_DIS
LIN {X -107.0877,Y 88.4181,Z 173,A 141.9876,B 8.249,C 0.1546,E1 8.1267,E2 309.7777} C_DIS
LIN {X -110.9879,Y 83.4699,Z 173,A 144.3534,B 8.2488,C 0.1643,E1 8.1227,E2 307.4438} C_DIS
LIN {X -112.7247,Y 81.1098,Z 173,A 145.8816,B 8.2488,C 0.1622,E1 8.1201,E2 305.8767} C_DIS
LIN {X -115.2826,Y 77.431,Z 173,A 147.7101,B 8.2488,C 0.1669,E1 8.1172,E2 304.0526} C_DIS
LIN {X -118.6833,Y 72.11,Z 173,A 150.3873,B 8.2487,C 0.1722,E1 8.1132,E2 301.3691} C_DIS
LIN {X -121.3184,Y 67.5815,Z 173,A 152.4434,B 8.2485,C 0.1793,E1 8.1104,E2 299.3284} C_DIS
LIN {X -123.0792,Y 64.3157,Z 173,A 154.0283,B 8.2485,C 0.1824,E1 8.1083,E2 297.7382} C_DIS
LIN {X -124.6209,Y 61.2749,Z 173,A 155.493,B 8.2484,C 0.1852,E1 8.1065,E2 296.2676} C_DIS
LIN {X -126.3372,Y 57.6571,Z 173,A 157.132,B 8.2483,C 0.1898,E1 8.1045,E2 294.632} C_DIS
LIN {X -127.5455,Y 54.9285,Z 173,A 158.4124,B 8.2483,C 0.1923,E1 8.1031,E2 293.3465} C_DIS
LIN {X -128.8672,Y 51.7517,Z 173,A 159.8591,B 8.2481,C 0.1957,E1 8.1016,E2 291.8978} C_DIS
LIN {X -130.2859,Y 48.073,Z 173,A 161.4642,B 8.2481,C 0.2005,E1 8.1,E2 290.2972} C_DIS
LIN {X -131.28,Y 45.2833,Z 173,A 162.7281,B 8.248,C 0.2032,E1 8.0988,E2 289.0291} C_DIS
LIN {X -132.3867,Y 41.9387,Z 173,A 164.1966,B 8.2479,C 0.2069,E1 8.0976,E2 287.5602} C_DIS
LIN {X -133.3757,Y 38.6786,Z 173,A 165.6411,B 8.2478,C 0.2103,E1 8.0964,E2 286.1121} C_DIS
LIN {X -134.2085,Y 35.6804,Z 173,A 166.963,B 8.2478,C 0.2133,E1 8.0954,E2 284.7867} C_DIS
LIN {X -135.1273,Y 32.0296,Z 173,A 168.4745,B 8.2476,C 0.2183,E1 8.0944,E2 283.282} C_DIS
LIN {X -135.7763,Y 29.1521,Z 173,A 170.626,B 8.2479,C 0.2076,E1 8.0932,E2 281.0128} C_DIS
LIN {X -136.957,Y 22.9745,Z 173,A 172.14,B 8.2472,C 0.2314,E1 8.0925,E2 279.6389} C_DIS
LIN {X -137.3423,Y 20.5577,Z 173,A 173.5748,B 8.2473,C 0.2279,E1 8.0918,E2 278.1514} C_DIS
LIN {X -137.8803,Y 16.5559,Z 173,A 175.5476,B 8.2473,C 0.228,E1 8.0912,E2 276.1411} C_DIS
LIN {X -138.3053,Y 12.54,Z 173,A 176.807,B 8.247,C 0.239,E1 8.0908,E2 274.935} C_DIS
LIN {X -138.5182,Y 9.8909,Z 173,A 178.3815,B 8.2471,C 0.2349,E1 8.0905,E2 273.3007} C_DIS
LIN {X -138.7484,Y 5.8436,Z 173,A 179.7206,B 8.2468,C 0.2448,E1 8.0904,E2 272.0057} C_DIS
LIN {X -138.8548,Y 2.1169,Z 173,A -178.3241,B 8.2468,C 0.2429,E1 8.0903,E2 269.9985} C_DIS
LIN {X -138.856,Y -2.0424,Z 173,A -176.8252,B 8.2466,C 0.2512,E1 8.0903,E2 268.529} C_DIS
LIN {X -138.683,Y -7.2227,Z 173,A -174.917,B 8.2464,C 0.2608,E1 8.0905,E2 266.6519} C_DIS
LIN {X -138.4974,Y -10.1763,Z 173,A -173.6018,B 8.2463,C 0.2629,E1 8.0908,E2 265.3258} C_DIS
LIN {X -137.8816,Y -16.545,Z 173,A -170.9076,B 8.2461,C 0.2697,E1 8.0916,E2 262.6271} C_DIS
LIN {X -137.4002,Y -20.162,Z 173,A -169.3741,B 8.2459,C 0.2735,E1 8.0921,E2 261.0912} C_DIS
LIN {X -136.7295,Y -24.2919,Z 173,A -167.5795,B 8.2459,C 0.2774,E1 8.093,E2 259.2893} C_DIS
LIN {X -136.034,Y -27.9254,Z 173,A -166.1041,B 8.2456,C 0.2825,E1 8.0938,E2 257.8216} C_DIS
LIN {X -135.3007,Y -31.2868,Z 173,A -164.6236,B 8.2456,C 0.2855,E1 8.0947,E2 256.3344} C_DIS
LIN {X -134.4049,Y -34.9425,Z 173,A -162.9073,B 8.2455,C 0.2873,E1 8.0959,E2 254.5984} C_DIS
LIN {X -133.2762,Y -39.0185,Z 173,A -161.2743,B 8.2452,C 0.2939,E1 8.0971,E2 252.981} C_DIS
LIN {X -132.2166,Y -42.4712,Z 173,A -159.7138,B 8.2452,C 0.2968,E1 8.0984,E2 251.4126} C_DIS
LIN {X -130.0767,Y -48.6315,Z 173,A -157.3148,B 8.2447,C 0.3086,E1 8.1007,E2 249.0527} C_DIS
LIN {X -128.5258,Y -52.5987,Z 173,A -155.2578,B 8.2447,C 0.3086,E1 8.1028,E2 246.9588} C_DIS
LIN {X -127.422,Y -55.214,Z 173,A -154.0718,B 8.2447,C 0.3115,E1 8.1041,E2 245.7716} C_DIS
LIN {X -125.9311,Y -58.5352,Z 173,A -152.4969,B 8.2445,C 0.3143,E1 8.1059,E2 244.1883} C_DIS
LIN {X -124.3531,Y -61.8177,Z 173,A -150.9556,B 8.2444,C 0.3175,E1 8.1078,E2 242.6429} C_DIS
LIN {X -121.5398,Y -67.1831,Z 173,A -148.3802,B 8.2442,C 0.3226,E1 8.1112,E2 240.0593} C_DIS
LIN {X -119.1926,Y -71.2647,Z 173,A -146.418,B 8.244,C 0.327,E1 8.114,E2 238.0957} C_DIS
LIN {X -116.8123,Y -75.103,Z 173,A -144.4706,B 8.2439,C 0.3301,E1 8.1169,E2 236.1384} C_DIS
LIN {X -114.7261,Y -78.2533,Z 173,A -142.9147,B 8.2437,C 0.3338,E1 8.1193,E2 234.5836} C_DIS
LIN {X -112.1672,Y -81.8792,Z 173,A -141.0208,B 8.2437,C 0.337,E1 8.1224,E2 232.6825} C_DIS
LIN {X -109.3824,Y -85.5632,Z 173,A -139.0952,B 8.2434,C 0.3409,E1 8.1257,E2 230.7551} C_DIS
LIN {X -106.5391,Y -89.0785,Z 173,A -137.2096,B 8.2433,C 0.3447,E1 8.1291,E2 228.8677} C_DIS
LIN {X -101.2713,Y -95.025,Z 173,A -134.1892,B 8.2428,C 0.3557,E1 8.1347,E2 225.8818} C_DIS
LIN {X -99.3008,Y -97.0819,Z 173,A -132.4388,B 8.2431,C 0.3486,E1 8.1382,E2 224.0573} C_DIS
LIN {X -96.6352,Y -99.7353,Z 173,A -131.2269,B 8.2428,C 0.3572,E1 8.1405,E2 222.89} C_DIS
LIN {X -93.7123,Y -102.4872,Z 173,A -129.4576,B 8.2428,C 0.3585,E1 8.1442,E2 221.1065} C_DIS
LIN {X -90.2698,Y -105.5322,Z 173,A -127.5201,B 8.2426,C 0.3612,E1 8.1483,E2 219.1641} C_DIS
LIN {X -86.7083,Y -108.477,Z 173,A -125.603,B 8.2425,C 0.3644,E1 8.1524,E2 217.246} C_DIS
LIN {X -83.0288,Y -111.3181,Z 173,A -122.8818,B 8.2429,C 0.354,E1 8.1588,E2 214.4201} C_DIS
LIN {X -77.6079,Y -115.1633,Z 173,A -121.1747,B 8.2419,C 0.3758,E1 8.1624,E2 212.8487} C_DIS
LIN {X -73.8365,Y -117.6171,Z 173,A -119.072,B 8.242,C 0.3743,E1 8.1674,E2 210.7143} C_DIS
LIN {X -70.0961,Y -119.8837,Z 173,A -117.2224,B 8.242,C 0.3761,E1 8.1718,E2 208.8588} C_DIS
LIN {X -62.0118,Y -124.2573,Z 173,A -113.5836,B 8.2416,C 0.3835,E1 8.1808,E2 205.2403} C_DIS
LIN {X -57.5467,Y -126.3882,Z 173,A -111.251,B 8.2417,C 0.3807,E1 8.1868,E2 202.8697} C_DIS
LIN {X -53.3771,Y -128.2024,Z 173,A -109.4985,B 8.2415,C 0.3848,E1 8.1912,E2 201.1331} C_DIS
LIN {X -49.9136,Y -129.5908,Z 173,A -107.9922,B 8.2415,C 0.3868,E1 8.1951,E2 199.631} C_DIS
LIN {X -46.8268,Y -130.7375,Z 173,A -106.6465,B 8.2414,C 0.3883,E1 8.1987,E2 198.2868} C_DIS
LIN {X -43.5634,Y -131.861,Z 173,A -105.2304,B 8.2414,C 0.3896,E1 8.2024,E2 196.8715} C_DIS
LIN {X -40.0272,Y -132.9783,Z 173,A -103.6999,B 8.2413,C 0.3907,E1 8.2065,E2 195.3406} C_DIS
LIN {X -37.0732,Y -133.8308,Z 173,A -101.8507,B 8.2417,C 0.3811,E1 8.2117,E2 193.4151} C_DIS
LIN {X -32.5117,Y -135.0111,Z 173,A -99.9355,B 8.2417,C 0.3827,E1 8.2169,E2 191.5032} C_DIS
LIN {X -28.0502,Y -136.0086,Z 173,A -98.7399,B 8.241,C 0.3961,E1 8.2199,E2 190.3976} C_DIS
LIN {X -21.3544,Y -137.219,Z 173,A -96.0207,B 8.2409,C 0.3989,E1 8.2274,E2 187.6891} C_DIS
LIN {X -16.545,Y -137.8816,Z 173,A -93.7166,B 8.2411,C 0.3939,E1 8.2338,E2 185.3451} C_DIS
LIN {X -12.7496,Y -138.2852,Z 173,A -92.1955,B 8.2411,C 0.3951,E1 8.238,E2 183.8305} C_DIS
LIN {X -8.9069,Y -138.5853,Z 173,A -90.5402,B 8.2411,C 0.394,E1 8.2427,E2 182.1659} C_DIS
LIN {X -5.3359,Y -138.7682,Z 173,A -89.1249,B 8.2411,C 0.3952,E1 8.2466,E2 180.7579} C_DIS
LIN {X -2.0027,Y -138.8567,Z 173,A -87.7392,B 8.2411,C 0.3949,E1 8.2505,E2 179.3703} C_DIS
LIN {X 0.9819,Y -138.8672,Z 173,A -87.0069,B 8.2406,C 0.4041,E1 8.2524,E2 178.7024} C_DIS
Enddeposition()
LIN {X 0.9819,Y -138.8672,Z 173,A -87.0069,B 8.2406,C 0.4041,E1 8.2524,E2 178.7024} C_DIS
Startdeposition()
$VEL.CP = VEL_PRINT
LIN {X 0.4042,Y -139.7793,Z 173,A -87.3658,B 8.08,C 0.413,E1 8.0911,E2 179.1577} C_DIS
LIN {X -3.8332,Y -139.7268,Z 173,A -89.0497,B 8.08,C 0.4121,E1 8.0864,E2 180.8354} C_DIS
LIN {X -8.2029,Y -139.5389,Z 173,A -90.8272,B 8.0801,C 0.4118,E1 8.0815,E2 182.6117} C_DIS
LIN {X -12.1249,Y -139.2528,Z 173,A -92.5337,B 8.0801,C 0.4134,E1 8.0767,E2 184.3312} C_DIS
LIN {X -16.4645,Y -138.8061,Z 173,A -94.2567,B 8.0801,C 0.4118,E1 8.0719,E2 186.0463} C_DIS
LIN {X -20.6601,Y -138.2458,Z 173,A -95.9848,B 8.0801,C 0.4112,E1 8.0672,E2 187.7743} C_DIS
LIN {X -26.8491,Y -137.1776,Z 173,A -98.6176,B 8.0801,C 0.4112,E1 8.0599,E2 190.4154} C_DIS
LIN {X -31.1378,Y -136.2667,Z 173,A -100.782,B 8.0799,C 0.4168,E1 8.0539,E2 192.6278} C_DIS
LIN {X -35.349,Y -135.2366,Z 173,A -102.3677,B 8.0801,C 0.4124,E1 8.0496,E2 194.1892} C_DIS
LIN {X -38.501,Y -134.3744,Z 173,A -103.5261,B 8.0803,C 0.4083,E1 8.0466,E2 195.3244} C_DIS
LIN {X -42.2593,Y -133.238,Z 173,A -105.0522,B 8.0804,C 0.4057,E1 8.0425,E2 196.84} C_DIS
LIN {X -45.5709,Y -132.1419,Z 173,A -106.4653,B 8.0804,C 0.4042,E1 8.0388,E2 198.2512} C_DIS
LIN {X -48.4963,Y -131.0975,Z 173,A -107.87,B 8.0804,C 0.4054,E1 8.0351,E2 199.6731} C_DIS
LIN {X -52.3589,Y -129.602,Z 173,A -109.4637,B 8.0806,C 0.402,E1 8.031,E2 201.2534} C_DIS
LIN {X -55.2609,Y -128.3916,Z 173,A -110.5706,B 8.0808,C 0.3975,E1 8.0282,E2 202.3368} C_DIS
LIN {X -59.4715,Y -126.499,Z 173,A -112.696,B 8.0808,C 0.3995,E1 8.0227,E2 204.4927} C_DIS
LIN {X -68.8011,Y -121.6766,Z 173,A -117.1499,B 8.0808,C 0.3967,E1 8.0117,E2 208.9661} C_DIS
LIN {X -72.7417,Y -119.3628,Z 173,A -118.9477,B 8.081,C 0.3928,E1 8.0074,E2 210.754} C_DIS
LIN {X -76.8815,Y -116.7386,Z 173,A -121.0217,B 8.0811,C 0.3909,E1 8.0025,E2 212.8362} C_DIS
LIN {X -83.3684,Y -112.198,Z 173,A -124.3363,B 8.0813,C 0.3869,E1 7.9949,E2 216.1593} C_DIS
LIN {X -87.0995,Y -109.3267,Z 173,A -126.2762,B 8.0815,C 0.3838,E1 7.9906,E2 218.1002} C_DIS
LIN {X -90.7427,Y -106.3226,Z 173,A -128.2414,B 8.0816,C 0.3809,E1 7.9864,E2 220.0688} C_DIS
LIN {X -94.0251,Y -103.4309,Z 173,A -130.0439,B 8.0818,C 0.3777,E1 7.9827,E2 221.8721} C_DIS
LIN {X -96.7602,Y -100.8771,Z 173,A -132.1793,B 8.0815,C 0.3844,E1 7.9782,E2 224.0842} C_DIS
LIN {X -100.5746,Y -97.0745,Z 173,A -134.8849,B 8.0813,C 0.3877,E1 7.9729,E2 226.8521} C_DIS
LIN {X -105.9154,Y -91.2173,Z 173,A -137.1053,B 8.0824,C 0.3648,E1 7.969,E2 228.9404} C_DIS
LIN {X -108.7795,Y -87.782,Z 173,A -138.9833,B 8.0824,C 0.3615,E1 7.9657,E2 230.8235} C_DIS
LIN {X -111.5868,Y -84.1845,Z 173,A -140.8802,B 8.0827,C 0.3578,E1 7.9624,E2 232.723} C_DIS
LIN {X -114.3366,Y -80.4105,Z 173,A -142.7834,B 8.0829,C 0.3532,E1 7.9593,E2 234.6239} C_DIS
LIN {X -116.8299,Y -76.7427,Z 173,A -144.4592,B 8.0831,C 0.3468,E1 7.9568,E2 236.2805} C_DIS
LIN {X -118.7968,Y -73.6617,Z 173,A -146.1634,B 8.0831,C 0.3464,E1 7.9542,E2 238.0104} C_DIS
LIN {X -121.6523,Y -68.8415,Z 173,A -149.0309,B 8.0831,C 0.3494,E1 7.9501,E2 240.9494} C_DIS
LIN {X -124.0249,Y -64.4689,Z 173,A -150.6395,B 8.0835,C 0.3378,E1 7.9481,E2 242.5021} C_DIS
LIN {X -125.9873,Y -60.5425,Z 173,A -152.3491,B 8.0838,C 0.3318,E1 7.946,E2 244.1992} C_DIS
LIN {X -127.4387,Y -57.4251,Z 173,A -153.762,B 8.0839,C 0.3282,E1 7.9443,E2 245.6116} C_DIS
LIN {X -129.0673,Y -53.6637,Z 173,A -155.7127,B 8.0839,C 0.3279,E1 7.9422,E2 247.5958} C_DIS
LIN {X -130.9075,Y -49.0035,Z 173,A -157.9883,B 8.084,C 0.3258,E1 7.9399,E2 249.8981} C_DIS
LIN {X -132.3121,Y -45.08,Z 173,A -159.4338,B 8.0843,C 0.3172,E1 7.9386,E2 251.3092} C_DIS
LIN {X -133.5905,Y -41.1313,Z 173,A -160.9901,B 8.0846,C 0.3104,E1 7.9373,E2 252.8457} C_DIS
LIN {X -134.5325,Y -37.9375,Z 173,A -162.3772,B 8.0847,C 0.307,E1 7.9362,E2 254.2347} C_DIS
LIN {X -135.4245,Y -34.6182,Z 173,A -163.8897,B 8.0848,C 0.3046,E1 7.9352,E2 255.7593} C_DIS
LIN {X -136.2421,Y -31.2456,Z 173,A -165.3608,B 8.085,C 0.3014,E1 7.9342,E2 257.2356} C_DIS
LIN {X -137.1583,Y -26.9498,Z 173,A -167.1147,B 8.0852,C 0.2956,E1 7.9332,E2 258.9821} C_DIS
LIN {X -137.8278,Y -23.276,Z 173,A -168.7288,B 8.0852,C 0.2925,E1 7.9324,E2 260.6056} C_DIS
LIN {X -138.3806,Y -19.7236,Z 173,A -170.1974,B 8.0854,C 0.2883,E1 7.9318,E2 262.0724} C_DIS
LIN {X -139.0689,Y -14.0792,Z 173,A -172.8514,B 8.0854,C 0.2864,E1 7.931,E2 264.7653} C_DIS
LIN {X -139.3648,Y -10.7725,Z 173,A -174.0474,B 8.0857,C 0.28,E1 7.9307,E2 265.9394} C_DIS
LIN {X -139.7192,Y -4.1038,Z 173,A -176.5033,B 8.0861,C 0.268,E1 7.9304,E2 268.3572} C_DIS
LIN {X -139.7497,Y 2.9463,Z 173,A -179.6353,B 8.0863,C 0.2633,E1 7.9304,E2 271.5175} C_DIS
LIN {X -139.413,Y 10.1123,Z 173,A 177.4722,B 8.0866,C 0.2541,E1 7.9308,E2 274.4014} C_DIS
LIN {X -138.7374,Y 17.0406,Z 173,A 174.3366,B 8.0866,C 0.25,E1 7.9317,E2 277.5701} C_DIS
LIN {X -138.2686,Y 20.5072,Z 173,A 172.732,B 8.0867,C 0.2484,E1 7.9324,E2 279.1949} C_DIS
LIN {X -137.5113,Y 25.0796,Z 173,A 170.8374,B 8.0869,C 0.2429,E1 7.9333,E2 281.087} C_DIS
LIN {X -136.4602,Y 30.2896,Z 173,A 168.7074,B 8.0871,C 0.2361,E1 7.9345,E2 283.2089} C_DIS
LIN {X -135.5397,Y 34.1643,Z 173,A 167.2059,B 8.0873,C 0.2295,E1 7.9355,E2 284.6923} C_DIS
LIN {X -134.6671,Y 37.4563,Z 173,A 165.7746,B 8.0873,C 0.2261,E1 7.9365,E2 286.1266} C_DIS
LIN {X -133.853,Y 40.2736,Z 173,A 164.3994,B 8.0874,C 0.2253,E1 7.9376,E2 287.5224} C_DIS
LIN {X -132.7091,Y 43.8921,Z 173,A 163.0021,B 8.0876,C 0.2187,E1 7.9388,E2 288.8983} C_DIS
LIN {X -131.5143,Y 47.3512,Z 173,A 161.4069,B 8.0876,C 0.216,E1 7.9403,E2 290.5039} C_DIS
LIN {X -130.2761,Y 50.6584,Z 173,A 159.8509,B 8.0877,C 0.2137,E1 7.9418,E2 292.0722} C_DIS
LIN {X -128.6423,Y 54.681,Z 173,A 158.0265,B 8.0878,C 0.2096,E1 7.9438,E2 293.9005} C_DIS
LIN {X -127.0568,Y 58.2655,Z 173,A 156.4525,B 8.088,C 0.2048,E1 7.9456,E2 295.4687} C_DIS
LIN {X -125.6779,Y 61.1857,Z 173,A 155.0203,B 8.088,C 0.203,E1 7.9473,E2 296.9132} C_DIS
LIN {X -123.8936,Y 64.719,Z 173,A 153.4651,B 8.0881,C 0.1978,E1 7.9493,E2 298.4584} C_DIS
LIN {X -122.3453,Y 67.6041,Z 173,A 151.9549,B 8.0881,C 0.1969,E1 7.9514,E2 299.9883} C_DIS
LIN {X -120.1378,Y 71.4534,Z 173,A 150.1825,B 8.0883,C 0.1916,E1 7.9538,E2 301.7531} C_DIS
LIN {X -117.0509,Y 76.4059,Z 173,A 147.7388,B 8.0883,C 0.1865,E1 7.9575,E2 304.2008} C_DIS
LIN {X -114.6332,Y 79.987,Z 173,A 145.9164,B 8.0885,C 0.183,E1 7.9604,E2 306.0279} C_DIS
LIN {X -112.0221,Y 83.6046,Z 173,A 144.1218,B 8.0885,C 0.1782,E1 7.9633,E2 307.8164} C_DIS
LIN {X -109.0696,Y 87.4224,Z 173,A 142.0472,B 8.0886,C 0.1752,E1 7.9669,E2 309.9012} C_DIS
LIN {X -104.4655,Y 92.8751,Z 173,A 138.4743,B 8.0886,C 0.1785,E1 7.9736,E2 313.5514} C_DIS
LIN {X -100.6421,Y 97.0048,Z 173,A 136.7443,B 8.0889,C 0.1649,E1 7.9768,E2 315.2079} C_DIS
LIN {X -94.8538,Y 102.6719,Z 173,A 132.8407,B 8.0889,C 0.1672,E1 7.9848,E2 319.1805} C_DIS
LIN {X -90.9086,Y 106.1812,Z 173,A 131.1821,B 8.089,C 0.1552,E1 7.9882,E2 320.7746} C_DIS
LIN {X -88.3729,Y 108.3,Z 173,A 129.4335,B 8.089,C 0.1589,E1 7.9921,E2 322.5708} C_DIS
LIN {X -84.9024,Y 111.0413,Z 173,A 127.9821,B 8.0891,C 0.15,E1 7.9952,E2 323.9759} C_DIS
LIN {X -81.0005,Y 113.9198,Z 173,A 125.9905,B 8.0892,C 0.1467,E1 7.9997,E2 325.9662} C_DIS
LIN {X -77.4466,Y 116.3646,Z 173,A 124.4486,B 8.0893,C 0.1402,E1 8.0032,E2 327.4784} C_DIS
LIN {X -74.0996,Y 118.5242,Z 173,A 122.5358,B 8.0893,C 0.1421,E1 8.0078,E2 329.4247} C_DIS
LIN {X -67.4113,Y 122.452,Z 173,A 119.3982,B 8.0893,C 0.1368,E1 8.0154,E2 332.5545} C_DIS
LIN {X -63.9101,Y 124.3137,Z 173,A 117.7635,B 8.0894,C 0.1348,E1 8.0194,E2 334.189} C_DIS
LIN {X -61.4966,Y 125.5245,Z 173,A 116.116,B 8.0893,C 0.1421,E1 8.0237,E2 335.9025} C_DIS
LIN {X -57.1278,Y 127.5716,Z 173,A 114.6663,B 8.0895,C 0.1311,E1 8.0272,E2 337.2854} C_DIS
LIN {X -53.7445,Y 129.0336,Z 173,A 112.852,B 8.0895,C 0.1344,E1 8.032,E2 339.1362} C_DIS
LIN {X -50.5029,Y 130.3365,Z 173,A 112.1066,B 8.0896,C 0.1216,E1 8.0337,E2 339.7951} C_DIS
LIN {X -44.9355,Y 132.3616,Z 173,A 109.1383,B 8.0896,C 0.1281,E1 8.0417,E2 342.8292} C_DIS
LIN {X -41.2404,Y 133.5571,Z 173,A 107.6973,B 8.0896,C 0.1242,E1 8.0454,E2 344.2503} C_DIS
LIN {X -37.8875,Y 134.5465,Z 173,A 106.2516,B 8.0896,C 0.1233,E1 8.0493,E2 345.6967} C_DIS
LIN {X -33.6874,Y 135.6608,Z 173,A 104.3549,B 8.0896,C 0.1239,E1 8.0545,E2 347.6066} C_DIS
LIN {X -29.0775,Y 136.7218,Z 173,A 102.3804,B 8.0896,C 0.1233,E1 8.0599,E2 349.5842} C_DIS
LIN {X -25.0349,Y 137.5195,Z 173,A 100.1252,B 8.0895,C 0.1319,E1 8.0663,E2 351.9083} C_DIS
LIN {X -19.6173,Y 138.3958,Z 173,A 98.5253,B 8.0896,C 0.1199,E1 8.0705,E2 353.4266} C_DIS
LIN {X -15.6635,Y 138.9006,Z 173,A 96.9794,B 8.0896,C 0.1178,E1 8.0747,E2 354.9608} C_DIS
LIN {X -10.7901,Y 139.3635,Z 173,A 94.8194,B 8.0896,C 0.12,E1 8.0808,E2 357.1388} C_DIS
LIN {X -5.2,Y 139.6828,Z 173,A 92.6292,B 8.0896,C 0.1178,E1 8.0868,E2 359.3149} C_DIS
LIN {X -1.1162,Y 139.7753,Z 173,A 91.0433,B 8.0896,C 0.1161,E1 8.0912,E2 360.8889} C_DIS
LIN {X 2.3363,Y 139.7598,Z 173,A 89.2634,B 8.0896,C 0.1226,E1 8.0963,E2 362.7135} C_DIS
LIN {X 8.7365,Y 139.506,Z 173,A 86.824,B 8.0896,C 0.1196,E1 8.1031,E2 365.1288} C_DIS
LIN {X 13.0377,Y 139.1702,Z 173,A 85.2452,B 8.0896,C 0.1167,E1 8.1074,E2 366.6832} C_DIS
LIN {X 17.3533,Y 138.7001,Z 173,A 83.2477,B 8.0896,C 0.1212,E1 8.113,E2 368.7074} C_DIS
LIN {X 24.2377,Y 137.6622,Z 173,A 80.5531,B 8.0896,C 0.1195,E1 8.1204,E2 371.3812} C_DIS
LIN {X 32.289,Y 135.9993,Z 173,A 76.9666,B 8.0896,C 0.1255,E1 8.1303,E2 374.9939} C_DIS
LIN {X 37.206,Y 134.7371,Z 173,A 75.0891,B 8.0896,C 0.1233,E1 8.1353,E2 376.8456} C_DIS
LIN {X 40.5971,Y 133.754,Z 173,A 73.6242,B 8.0896,C 0.1248,E1 8.1392,E2 378.3125} C_DIS
LIN {X 44.2168,Y 132.601,Z 173,A 72.0754,B 8.0896,C 0.126,E1 8.1433,E2 379.86} C_DIS
LIN {X 47.6216,Y 131.4168,Z 173,A 70.6202,B 8.0896,C 0.127,E1 8.1471,E2 381.3122} C_DIS
LIN {X 51.1023,Y 130.1035,Z 173,A 69.0914,B 8.0896,C 0.1286,E1 8.1511,E2 382.8414} C_DIS
LIN {X 56.6616,Y 127.7802,Z 173,A 66.7951,B 8.0896,C 0.1281,E1 8.157,E2 385.1157} C_DIS
LIN {X 63.9029,Y 124.3174,Z 173,A 63.2479,B 8.0894,C 0.1371,E1 8.166,E2 388.6952} C_DIS
LIN {X 68.1907,Y 122.0197,Z 173,A 61.2992,B 8.0894,C 0.139,E1 8.1707,E2 390.6384} C_DIS
LIN {X 71.7486,Y 119.9619,Z 173,A 59.6223,B 8.0894,C 0.1413,E1 8.1747,E2 392.3144} C_DIS
LIN {X 75.7672,Y 117.4656,Z 173,A 57.8296,B 8.0894,C 0.1414,E1 8.1789,E2 394.0889} C_DIS
LIN {X 80.7017,Y 114.1311,Z 173,A 55.3284,B 8.0892,C 0.1465,E1 8.1847,E2 396.5979} C_DIS
LIN {X 84.4063,Y 111.4195,Z 173,A 53.5041,B 8.0892,C 0.1486,E1 8.1888,E2 398.4153} C_DIS
LIN {X 87.8229,Y 108.7465,Z 173,A 51.747,B 8.0892,C 0.1514,E1 8.1926,E2 400.1701} C_DIS
LIN {X 91.1103,Y 106.0075,Z 173,A 50.1649,B 8.0892,C 0.1512,E1 8.196,E2 401.731} C_DIS
LIN {X 93.6486,Y 103.7725,Z 173,A 48.641,B 8.089,C 0.1566,E1 8.1992,E2 403.2726} C_DIS
LIN {X 98.111,Y 99.564,Z 173,A 46.0929,B 8.089,C 0.1622,E1 8.2043,E2 405.8257} C_DIS
LIN {X 101.3675,Y 96.247,Z 173,A 44.4735,B 8.089,C 0.1604,E1 8.2074,E2 407.4095} C_DIS
LIN {X 104.6891,Y 92.6221,Z 173,A 42.2714,B 8.0888,C 0.1685,E1 8.2116,E2 409.6361} C_DIS
LIN {X 107.5281,Y 89.3108,Z 173,A 40.1783,B 8.0886,C 0.1785,E1 8.2154,E2 411.7683} C_DIS
LIN {X 109.9664,Y 86.2899,Z 173,A 38.8326,B 8.0886,C 0.1771,E1 8.2177,E2 413.0837} C_DIS
LIN {X 112.9398,Y 82.3615,Z 173,A 36.9024,B 8.0886,C 0.18,E1 8.2209,E2 415.0036} C_DIS
LIN {X 115.4673,Y 78.7789,Z 173,A 35.1151,B 8.0884,C 0.184,E1 8.2237,E2 416.7904} C_DIS
LIN {X 117.9492,Y 75.0122,Z 173,A 33.3138,B 8.0884,C 0.1875,E1 8.2265,E2 418.5867} C_DIS
LIN {X 119.617,Y 72.3218,Z 173,A 31.4392,B 8.088,C 0.2025,E1 8.2293,E2 420.5345} C_DIS
LIN {X 122.4504,Y 67.4142,Z 173,A 29.7891,B 8.0882,C 0.1945,E1 8.2314,E2 422.1013} C_DIS
LIN {X 124.3953,Y 63.7498,Z 173,A 28.1677,B 8.0882,C 0.1972,E1 8.2335,E2 423.7135} C_DIS
LIN {X 127.2792,Y 57.7816,Z 173,A 25.537,B 8.088,C 0.2025,E1 8.2366,E2 426.335} C_DIS
LIN {X 129.9957,Y 51.3795,Z 173,A 22.7071,B 8.0878,C 0.2096,E1 8.2397,E2 429.1642} C_DIS
LIN {X 131.4304,Y 47.5837,Z 173,A 21.1038,B 8.0878,C 0.2128,E1 8.2412,E2 430.7609} C_DIS
LIN {X 132.6189,Y 44.1629,Z 173,A 19.6593,B 8.0877,C 0.216,E1 8.2425,E2 432.2013} C_DIS
LIN {X 133.5836,Y 41.1539,Z 173,A 18.3079,B 8.0875,C 0.2208,E1 8.2437,E2 433.5609} C_DIS
LIN {X 134.5935,Y 37.7194,Z 173,A 16.8711,B 8.0875,C 0.2242,E1 8.2448,E2 434.9948} C_DIS
LIN {X 135.4503,Y 34.5167,Z 173,A 15.5218,B 8.0873,C 0.2277,E1 8.2457,E2 436.3439} C_DIS
LIN {X 137.3544,Y 25.9244,Z 173,A 12.4357,B 8.0873,C 0.2269,E1 8.2476,E2 439.366} C_DIS
LIN {X 138.3443,Y 19.9777,Z 173,A 9.4497,B 8.0868,C 0.2449,E1 8.2489,E2 442.4203} C_DIS
LIN {X 139.1118,Y 13.6466,Z 173,A 7.0033,B 8.0868,C 0.2488,E1 8.2497,E2 444.8474} C_DIS
LIN {X 139.3767,Y 10.6098,Z 173,A 5.7358,B 8.0866,C 0.2528,E1 8.25,E2 446.1183} C_DIS
LIN {X 139.6059,Y 6.9607,Z 173,A 4.0431,B 8.0863,C 0.2612,E1 8.2502,E2 447.8371} C_DIS
LIN {X 139.7307,Y 3.6932,Z 173,A 2.7409,B 8.0863,C 0.2643,E1 8.2503,E2 449.1356} C_DIS
LIN {X 139.7809,Y 0.3544,Z 173,A 1.639,B 8.0863,C 0.2626,E1 8.2503,E2 450.2047} C_DIS
LIN {X 139.7331,Y -3.606,Z 173,A 0.0736,B 8.0862,C 0.266,E1 8.2503,E2 451.7639} C_DIS
LIN {X 139.5149,Y -8.5927,Z 173,A -1.9322,B 8.086,C 0.2711,E1 8.25,E2 453.7664} C_DIS
LIN {X 139.0259,Y -14.4995,Z 173,A -4.3607,B 8.0858,C 0.2781,E1 8.2494,E2 456.1972} C_DIS
LIN {X 138.6095,Y -18.0451,Z 173,A -5.7375,B 8.0857,C 0.2805,E1 8.2489,E2 457.5641} C_DIS
LIN {X 138.2255,Y -20.7911,Z 173,A -6.9646,B 8.0855,C 0.2857,E1 8.2484,E2 458.8041} C_DIS
LIN {X 137.5733,Y -24.7345,Z 173,A -8.5998,B 8.0854,C 0.2903,E1 8.2476,E2 460.4404} C_DIS
LIN {X 136.5197,Y -30.0138,Z 173,A -10.6659,B 8.0852,C 0.2936,E1 8.2465,E2 462.4905} C_DIS
LIN {X 135.236,Y -35.3534,Z 173,A -13.2807,B 8.0847,C 0.3076,E1 8.2447,E2 465.1543} C_DIS
LIN {X 134.2037,Y -39.084,Z 173,A -14.5355,B 8.0848,C 0.3051,E1 8.2437,E2 466.368} C_DIS
LIN {X 132.7867,Y -43.659,Z 173,A -16.4547,B 8.0846,C 0.3096,E1 8.2421,E2 468.2834} C_DIS
LIN {X 131.1833,Y -48.2674,Z 173,A -18.621,B 8.0843,C 0.3186,E1 8.24,E2 470.4732} C_DIS
LIN {X 129.998,Y -51.3736,Z 173,A -19.8199,B 8.0843,C 0.3189,E1 8.2388,E2 471.6523} C_DIS
LIN {X 128.4704,Y -55.0786,Z 173,A -21.1613,B 8.0843,C 0.3169,E1 8.2374,E2 472.9564} C_DIS
LIN {X 125.8395,Y -60.8519,Z 173,A -24.1169,B 8.0838,C 0.3313,E1 8.2339,E2 475.9606} C_DIS
LIN {X 123.2326,Y -65.9731,Z 173,A -26.2599,B 8.0838,C 0.333,E1 8.2312,E2 478.0785} C_DIS
LIN {X 121.0697,Y -69.8629,Z 173,A -28.0696,B 8.0835,C 0.3374,E1 8.2287,E2 479.8882} C_DIS
LIN {X 119.4264,Y -72.6369,Z 173,A -29.6198,B 8.0832,C 0.3455,E1 8.2264,E2 481.4693} C_DIS
LIN {X 117.4732,Y -75.7535,Z 173,A -30.8493,B 8.0832,C 0.3434,E1 8.2246,E2 482.6643} C_DIS
LIN {X 115.2247,Y -79.1323,Z 173,A -32.4628,B 8.0832,C 0.3465,E1 8.2221,E2 484.273} C_DIS
LIN {X 112.7729,Y -82.5891,Z 173,A -33.9968,B 8.0832,C 0.3464,E1 8.2196,E2 485.7824} C_DIS
LIN {X 108.722,Y -87.8533,Z 173,A -36.8788,B 8.0827,C 0.3561,E1 8.2146,E2 488.6879} C_DIS
LIN {X 105.6985,Y -91.4691,Z 173,A -38.6774,B 8.0827,C 0.3577,E1 8.2114,E2 490.471} C_DIS
LIN {X 102.2874,Y -95.2678,Z 173,A -41.0534,B 8.0822,C 0.3682,E1 8.2068,E2 492.8858} C_DIS
LIN {X 99.9066,Y -97.7617,Z 173,A -42.2433,B 8.0822,C 0.3666,E1 8.2046,E2 494.0482} C_DIS
LIN {X 96.7806,Y -100.8576,Z 173,A -44.0355,B 8.0822,C 0.3702,E1 8.201,E2 495.8406} C_DIS
LIN {X 92.5187,Y -104.7805,Z 173,A -46.6506,B 8.0817,C 0.3798,E1 8.1955,E2 498.4892} C_DIS
LIN {X 89.5521,Y -107.3276,Z 173,A -47.9601,B 8.0817,C 0.377,E1 8.1928,E2 499.7622} C_DIS
LIN {X 86.0689,Y -110.1405,Z 173,A -49.7691,B 8.0817,C 0.3799,E1 8.1888,E2 501.5695} C_DIS
LIN {X 81.902,Y -113.2729,Z 173,A -52.0346,B 8.0814,C 0.3864,E1 8.1837,E2 503.8537} C_DIS
LIN {X 77.2438,Y -116.5,Z 173,A -53.9231,B 8.0816,C 0.3816,E1 8.1795,E2 505.6877} C_DIS
LIN {X 74.4366,Y -118.3127,Z 173,A -55.9207,B 8.0809,C 0.3964,E1 8.1746,E2 507.7682} C_DIS
LIN {X 70.6209,Y -120.6292,Z 173,A -57.3735,B 8.0811,C 0.3918,E1 8.1712,E2 509.1736} C_DIS
LIN {X 66.7114,Y -122.8345,Z 173,A -59.1563,B 8.0811,C 0.3934,E1 8.1668,E2 510.9505} C_DIS
LIN {X 63.7038,Y -124.4188,Z 173,A -60.2559,B 8.0812,C 0.3896,E1 8.1642,E2 512.0128} C_DIS
LIN {X 60.4492,Y -126.0319,Z 173,A -61.8204,B 8.081,C 0.3931,E1 8.1603,E2 513.5884} C_DIS
LIN {X 58.2711,Y -127.0542,Z 173,A -63.5311,B 8.0803,C 0.4087,E1 8.1557,E2 515.3941} C_DIS
LIN {X 53.4683,Y -129.1489,Z 173,A -65.0568,B 8.0807,C 0.3992,E1 8.1519,E2 516.8408} C_DIS
LIN {X 49.8261,Y -130.5994,Z 173,A -66.621,B 8.0807,C 0.4002,E1 8.1479,E2 518.4008} C_DIS
LIN {X 47.2908,Y -131.536,Z 173,A -68.3155,B 8.0801,C 0.4128,E1 8.1432,E2 520.1722} C_DIS
LIN {X 42.5585,Y -133.1425,Z 173,A -69.7352,B 8.0806,C 0.4027,E1 8.1397,E2 521.5118} C_DIS
LIN {X 39.3874,Y -134.1149,Z 173,A -71.1097,B 8.0805,C 0.4043,E1 8.136,E2 522.8891} C_DIS
LIN {X 35.8351,Y -135.1075,Z 173,A -73.2909,B 8.0798,C 0.4184,E1 8.1299,E2 525.1583} C_DIS
LIN {X 30.4474,Y -136.4244,Z 173,A -74.9958,B 8.0802,C 0.4093,E1 8.1254,E2 526.7911} C_DIS
LIN {X 27.5235,Y -137.0429,Z 173,A -76.5453,B 8.0799,C 0.4163,E1 8.1211,E2 528.3835} C_DIS
LIN {X 23.3855,Y -137.8095,Z 173,A -77.753,B 8.0803,C 0.4076,E1 8.1179,E2 529.5251} C_DIS
LIN {X 16.7805,Y -138.7685,Z 173,A -80.5322,B 8.0803,C 0.4099,E1 8.1102,E2 532.3116} C_DIS
LIN {X 13.5021,Y -139.1256,Z 173,A -81.823,B 8.0803,C 0.4093,E1 8.1066,E2 533.5952} C_DIS
LIN {X 10.1408,Y -139.4109,Z 173,A -83.331,B 8.0801,C 0.4121,E1 8.1024,E2 535.1203} C_DIS
LIN {X 5.8719,Y -139.6566,Z 173,A -85.0576,B 8.0801,C 0.4121,E1 8.0976,E2 536.8445} C_DIS
LIN {X 2.2832,Y -139.7607,Z 173,A -86.5058,B 8.0801,C 0.4119,E1 8.0935,E2 538.2903} C_DIS
LIN {X 2.2832,Y -139.7607,Z 173,A -86.5058,B 8.0801,C 0.4119,E1 8.0935,E2 538.2903} C_DIS
Enddeposition()
LIN {X 0.9966,Y -140.684,Z 173,A -86.7228,B 8.0803,C 0.411,E1 8.0931,E2 538.5006} C_DIS
Startdeposition()
$VEL.CP = VEL_PRINT
LIN {X 5.3302,Y -140.5869,Z 173,A -84.5447,B 8.0807,C 0.4029,E1 8.0993,E2 536.2668} C_DIS
LIN {X 9.7591,Y -140.3497,Z 173,A -82.7343,B 8.0807,C 0.4023,E1 8.1044,E2 534.455} C_DIS
LIN {X 13.251,Y -140.0625,Z 173,A -81.4524,B 8.0807,C 0.4045,E1 8.1079,E2 533.1916} C_DIS
LIN {X 16.037,Y -139.7721,Z 173,A -80.3237,B 8.0807,C 0.4042,E1 8.111,E2 532.0638} C_DIS
LIN {X 19.8563,Y -139.2794,Z 173,A -78.5212,B 8.0809,C 0.3989,E1 8.1161,E2 530.2292} C_DIS
LIN {X 24.5999,Y -138.5204,Z 173,A -76.6993,B 8.0809,C 0.4004,E1 8.1211,E2 528.424} C_DIS
LIN {X 28.4372,Y -137.7842,Z 173,A -75.1288,B 8.0809,C 0.3997,E1 8.1254,E2 526.8553} C_DIS
LIN {X 32.3226,Y -136.9258,Z 173,A -73.4252,B 8.0809,C 0.3968,E1 8.13,E2 525.1396} C_DIS
LIN {X 37.1665,Y -135.6915,Z 173,A -71.4459,B 8.081,C 0.3962,E1 8.1354,E2 523.1665} C_DIS
LIN {X 41.2186,Y -134.5139,Z 173,A -69.8379,B 8.081,C 0.3968,E1 8.1396,E2 521.5718} C_DIS
LIN {X 45.3657,Y -133.1746,Z 173,A -68.0705,B 8.081,C 0.3951,E1 8.1443,E2 519.8043} C_DIS
LIN {X 48.892,Y -131.9195,Z 173,A -66.6511,B 8.081,C 0.3955,E1 8.148,E2 518.3976} C_DIS
LIN {X 52.2456,Y -130.6272,Z 173,A -65.0732,B 8.0812,C 0.3916,E1 8.1522,E2 516.8034} C_DIS
LIN {X 59.4615,Y -127.5047,Z 173,A -61.9127,B 8.0814,C 0.3883,E1 8.1602,E2 513.646} C_DIS
LIN {X 63.2889,Y -125.6495,Z 173,A -60.1021,B 8.0816,C 0.3844,E1 8.1648,E2 511.8236} C_DIS
LIN {X 66.9065,Y -123.7624,Z 173,A -58.4734,B 8.0816,C 0.3826,E1 8.1688,E2 510.1979} C_DIS
LIN {X 73.0013,Y -120.2678,Z 173,A -55.5911,B 8.0819,C 0.3778,E1 8.1758,E2 507.3104} C_DIS
LIN {X 76.8211,Y -117.8646,Z 173,A -53.8185,B 8.0819,C 0.3761,E1 8.1799,E2 505.5449} C_DIS
LIN {X 80.9971,Y -115.0346,Z 173,A -51.7391,B 8.0822,C 0.372,E1 8.1847,E2 503.4603} C_DIS
LIN {X 84.8341,Y -112.2349,Z 173,A -49.8908,B 8.0822,C 0.3703,E1 8.1888,E2 501.6217} C_DIS
LIN {X 87.896,Y -109.854,Z 173,A -48.2824,B 8.0824,C 0.3667,E1 8.1924,E2 500.0081} C_DIS
LIN {X 91.1781,Y -107.1449,Z 173,A -46.6486,B 8.0824,C 0.3654,E1 8.1958,E2 498.3858} C_DIS
LIN {X 94.2458,Y -104.4575,Z 173,A -44.8909,B 8.0827,C 0.3601,E1 8.1995,E2 496.6138} C_DIS
LIN {X 97.6084,Y -101.3223,Z 173,A -43.1053,B 8.0827,C 0.358,E1 8.2031,E2 494.8378} C_DIS
LIN {X 100.6019,Y -98.3503,Z 173,A -41.3627,B 8.083,C 0.3538,E1 8.2066,E2 493.0903} C_DIS
LIN {X 103.9756,Y -94.7769,Z 173,A -39.366,B 8.0832,C 0.3496,E1 8.2104,E2 491.0923} C_DIS
LIN {X 106.8663,Y -91.5053,Z 173,A -37.6749,B 8.0832,C 0.3474,E1 8.2135,E2 489.4109} C_DIS
LIN {X 109.6363,Y -88.1668,Z 173,A -35.7784,B 8.0835,C 0.3406,E1 8.2168,E2 487.4955} C_DIS
LIN {X 113.7728,Y -82.7605,Z 173,A -32.5545,B 8.0842,C 0.3243,E1 8.2223,E2 484.2085} C_DIS
LIN {X 117.0606,Y -78.0403,Z 173,A -31.1707,B 8.0836,C 0.3391,E1 8.2243,E2 482.9499} C_DIS
LIN {X 120.0293,Y -73.3926,Z 173,A -28.6994,B 8.084,C 0.3287,E1 8.228,E2 480.4467} C_DIS
LIN {X 122.1367,Y -69.8292,Z 173,A -26.9941,B 8.0842,C 0.324,E1 8.2304,E2 478.7371} C_DIS
LIN {X 124.2766,Y -65.944,Z 173,A -24.7626,B 8.0848,C 0.3102,E1 8.2334,E2 476.4473} C_DIS
LIN {X 126.4769,Y -61.6193,Z 173,A -23.3987,B 8.0844,C 0.3181,E1 8.235,E2 475.1627} C_DIS
LIN {X 128.1251,Y -58.1155,Z 173,A -21.7182,B 8.0847,C 0.3117,E1 8.237,E2 473.4669} C_DIS
LIN {X 129.527,Y -54.9205,Z 173,A -20.4549,B 8.0847,C 0.3113,E1 8.2384,E2 472.2231} C_DIS
LIN {X 131.0228,Y -51.245,Z 173,A -18.794,B 8.0849,C 0.3059,E1 8.2401,E2 470.5545} C_DIS
LIN {X 132.6129,Y -46.9825,Z 173,A -17.008,B 8.0851,C 0.3023,E1 8.2418,E2 468.7756} C_DIS
LIN {X 133.8909,Y -43.2011,Z 173,A -15.3214,B 8.0853,C 0.2965,E1 8.2433,E2 467.0793} C_DIS
LIN {X 135.8779,Y -36.472,Z 173,A -12.8259,B 8.0853,C 0.2963,E1 8.2452,E2 464.6287} C_DIS
LIN {X 136.7511,Y -33.0474,Z 173,A -11.1856,B 8.0856,C 0.2879,E1 8.2463,E2 462.9606} C_DIS
LIN {X 137.5157,Y -29.7058,Z 173,A -9.5345,B 8.0859,C 0.2784,E1 8.2473,E2 461.2745} C_DIS
LIN {X 138.1794,Y -26.4475,Z 173,A -8.5604,B 8.0858,C 0.2828,E1 8.2478,E2 460.3492} C_DIS
LIN {X 138.6743,Y -23.7232,Z 173,A -7.479,B 8.0858,C 0.2805,E1 8.2483,E2 459.2728} C_DIS
LIN {X 139.2419,Y -20.1188,Z 173,A -5.9171,B 8.086,C 0.2746,E1 8.249,E2 457.6995} C_DIS
LIN {X 139.6436,Y -17.1147,Z 173,A -4.8308,B 8.086,C 0.2743,E1 8.2494,E2 456.6315} C_DIS
LIN {X 140.0307,Y -13.5823,Z 173,A -3.2321,B 8.0863,C 0.2668,E1 8.2498,E2 455.0115} C_DIS
LIN {X 140.3495,Y -9.763,Z 173,A -1.7518,B 8.0863,C 0.2641,E1 8.2502,E2 453.5404} C_DIS
LIN {X 140.5632,Y -5.9381,Z 173,A -0.1932,B 8.0865,C 0.2596,E1 8.2504,E2 451.9805} C_DIS
LIN {X 140.6844,Y -1.1273,Z 173,A 1.8161,B 8.0867,C 0.2528,E1 8.2504,E2 449.963} C_DIS
LIN {X 140.6498,Y 3.3238,Z 173,A 3.5388,B 8.0868,C 0.2496,E1 8.2504,E2 448.2505} C_DIS
LIN {X 140.5341,Y 6.5909,Z 173,A 4.8195,B 8.0869,C 0.2468,E1 8.2502,E2 446.9753} C_DIS
LIN {X 140.3124,Y 10.271,Z 173,A 6.2718,B 8.087,C 0.2435,E1 8.25,E2 445.5281} C_DIS
LIN {X 139.9432,Y 14.4668,Z 173,A 8.0379,B 8.0872,C 0.2375,E1 8.2495,E2 443.754} C_DIS
LIN {X 139.2019,Y 20.399,Z 173,A 10.4006,B 8.0874,C 0.2321,E1 8.2486,E2 441.3987} C_DIS
LIN {X 138.5607,Y 24.3744,Z 173,A 11.9792,B 8.0874,C 0.2288,E1 8.2479,E2 439.8268} C_DIS
LIN {X 137.8919,Y 27.9077,Z 173,A 13.3764,B 8.0875,C 0.2261,E1 8.2472,E2 438.4372} C_DIS
LIN {X 137.24,Y 30.9566,Z 173,A 14.9753,B 8.0878,C 0.2155,E1 8.2462,E2 436.7943} C_DIS
LIN {X 136.4108,Y 34.4253,Z 173,A 15.8944,B 8.0876,C 0.2228,E1 8.2456,E2 435.9437} C_DIS
LIN {X 135.5667,Y 37.6127,Z 173,A 17.3886,B 8.0878,C 0.2158,E1 8.2445,E2 434.4288} C_DIS
LIN {X 134.7298,Y 40.5131,Z 173,A 18.701,B 8.0879,C 0.2107,E1 8.2434,E2 433.1048} C_DIS
LIN {X 133.3894,Y 44.7247,Z 173,A 20.4093,B 8.088,C 0.2077,E1 8.242,E2 431.4071} C_DIS
LIN {X 131.9078,Y 48.9232,Z 173,A 22.2152,B 8.0881,C 0.203,E1 8.2402,E2 429.601} C_DIS
LIN {X 130.8022,Y 51.8115,Z 173,A 23.7431,B 8.0884,C 0.1939,E1 8.2386,E2 428.0374} C_DIS
LIN {X 129.4135,Y 55.1867,Z 173,A 24.9865,B 8.0884,C 0.1952,E1 8.2373,E2 426.8246} C_DIS
LIN {X 127.8307,Y 58.7566,Z 173,A 26.3794,B 8.0884,C 0.1952,E1 8.2357,E2 425.4564} C_DIS
LIN {X 125.9139,Y 62.761,Z 173,A 28.3455,B 8.0885,C 0.1872,E1 8.2333,E2 423.4688} C_DIS
LIN {X 123.7435,Y 66.9417,Z 173,A 30.0582,B 8.0885,C 0.1866,E1 8.2311,E2 421.7817} C_DIS
Enddeposition()
END
